LIN {X 0,Y 418.667,Z 234.824,A -85,B 0,C 180,E1 -10080.004,E2 -10080.004} C_VEL
LIN {X 0,Y 418.499,Z 234.849,A -85,B 0,C 180,E1 -10082.892,E2 -10082.892} C_VEL
LIN {X 0,Y 418.499,Z 234.856,A -85,B 0,C 180,E1 -10085.787,E2 -10085.787} C_VEL
LIN {X 0,Y 418.397,Z 234.849,A -85,B 0,C 180,E1 -10088.699,E2 -10088.699} C_VEL
LIN {X 0,Y 418.316,Z 234.859,A -85,B 0,C 180,E1 -10091.635,E2 -10091.635} C_VEL
LIN {X 0,Y 418.306,Z 234.878,A -85,B 0,C 180,E1 -10094.601,E2 -10094.601} C_VEL
LIN {X 0,Y 418.29,Z 234.876,A -85,B 0,C 180,E1 -10097.607,E2 -10097.607} C_VEL
LIN {X 0,Y 418.255,Z 234.87,A -85,B 0,C 180,E1 -10100.666,E2 -10100.666} C_VEL
LIN {X 0,Y 418.28,Z 234.875,A -85,B 0,C 180,E1 -10103.785,E2 -10103.785} C_VEL
LIN {X 0,Y 418.317,Z 234.875,A -85,B 0,C 180,E1 -10107.073,E2 -10107.073} C_VEL
LIN {X 0,Y 418.251,Z 234.871,A -85,B 0,C 180,E1 -10110.275,E2 -10110.275} C_VEL
LIN {X 0,Y 418.24,Z 234.886,A -85,B 0,C 180,E1 -10113.681,E2 -10113.681} C_VEL
LIN {X 0,Y 418.246,Z 234.881,A -85,B 0,C 180,E1 -10117.227,E2 -10117.227} C_VEL
LIN {X 0,Y 418.237,Z 234.887,A -85,B 0,C 180,E1 -10119.687,E2 -10119.687} C_VEL
LIN {X 0,Y 418.232,Z 234.879,A -85,B 0,C 180,E1 -10122.322,E2 -10122.322} C_VEL
LIN {X 0,Y 418.245,Z 234.862,A -85,B 0,C 180,E1 -10125.111,E2 -10125.111} C_VEL
LIN {X 0,Y 418.243,Z 234.883,A -85,B 0,C 180,E1 -10127.768,E2 -10127.768} C_VEL
LIN {X 0,Y 418.247,Z 234.881,A -85,B 0,C 180,E1 -10131.558,E2 -10131.558} C_VEL
LIN {X 0,Y 418.269,Z 234.881,A -85,B 0,C 180,E1 -10135.16,E2 -10135.16} C_VEL
LIN {X 0,Y 418.255,Z 234.885,A -85,B 0,C 180,E1 -10137.473,E2 -10137.473} C_VEL
LIN {X 0,Y 418.279,Z 234.882,A -85,B 0,C 180,E1 -10140.897,E2 -10140.897} C_VEL
LIN {X 0,Y 418.338,Z 234.979,A -85,B 0,C 180,E1 -10143.833,E2 -10143.833} C_VEL
LIN {X 0,Y 419.166,Z 239.348,A -85,B 0,C 180,E1 -10144.881,E2 -10144.881} C_VEL
LIN {X 0,Y 420.709,Z 247.766,A -85,B 0,C 180,E1 -10146.753,E2 -10146.753} C_VEL
LIN {X 0,Y 420.134,Z 259.403,A -85,B 0,C 180,E1 -10149.178,E2 -10149.178} C_VEL
LIN {X 0,Y 419.569,Z 269.337,A -85,B 0,C 180,E1 -10151.189,E2 -10151.189} C_VEL
LIN {X 0,Y 420.301,Z 274.486,A -85,B 0,C 180,E1 -10151.353,E2 -10151.353} C_VEL
LIN {X 0,Y 423.345,Z 294.383,A -85,B 0,C 180,E1 -10151.82,E2 -10151.82} C_VEL
LIN {X 0,Y 422.372,Z 377.264,A -85,B 0,C 180,E1 -10153.258,E2 -10153.258} C_VEL
LIN {X 0,Y 421.886,Z 390.497,A -85,B 0,C 180,E1 -10153.674,E2 -10153.674} C_VEL
LIN {X 0,Y 421.378,Z 403.241,A -85,B 0,C 180,E1 -10154.275,E2 -10154.275} C_VEL
LIN {X 0,Y 420.699,Z 414.545,A -85,B 0,C 180,E1 -10154.993,E2 -10154.993} C_VEL
LIN {X 0,Y 419.998,Z 426.666,A -85,B 0,C 180,E1 -10155.999,E2 -10155.999} C_VEL
LIN {X 0,Y 419.321,Z 437.803,A -85,B 0,C 180,E1 -10157.169,E2 -10157.169} C_VEL
LIN {X 0,Y 418.652,Z 447.013,A -85,B 0,C 180,E1 -10158.379,E2 -10158.379} C_VEL
LIN {X 0,Y 418.063,Z 455.979,A -85,B 0,C 180,E1 -10159.834,E2 -10159.834} C_VEL
LIN {X 0,Y 417.61,Z 463.179,A -85,B 0,C 180,E1 -10161.289,E2 -10161.289} C_VEL
LIN {X 0,Y 417.295,Z 468.908,A -85,B 0,C 180,E1 -10162.744,E2 -10162.744} C_VEL
LIN {X 0,Y 417.132,Z 473.414,A -85,B 0,C 180,E1 -10164.198,E2 -10164.198} C_VEL
LIN {X 0,Y 417.119,Z 475.788,A -85,B 0,C 180,E1 -10165.168,E2 -10165.168} C_VEL
LIN {X 0,Y 417.003,Z 477.727,A -85,B 0,C 180,E1 -10166.135,E2 -10166.135} C_VEL
LIN {X 0,Y 416.988,Z 479.244,A -85,B 0,C 180,E1 -10167.102,E2 -10167.102} C_VEL
LIN {X 0,Y 417.034,Z 480.308,A -85,B 0,C 180,E1 -10168.069,E2 -10168.069} C_VEL
LIN {X 0,Y 416.987,Z 481.258,A -85,B 0,C 180,E1 -10170,E2 -10170} C_VEL
LIN {X 0,Y 416.997,Z 481.151,A -85,B 0,C 180,E1 -10170.966,E2 -10170.966} C_VEL
LIN {X 0,Y 417.035,Z 480.612,A -85,B 0,C 180,E1 -10171.932,E2 -10171.932} C_VEL
LIN {X 0,Y 417.005,Z 478.355,A -85,B 0,C 180,E1 -10173.866,E2 -10173.866} C_VEL
LIN {X 0,Y 417.164,Z 475.557,A -85,B 0,C 180,E1 -10175.317,E2 -10175.317} C_VEL
LIN {X 0,Y 417.253,Z 471.743,A -85,B 0,C 180,E1 -10176.771,E2 -10176.771} C_VEL
LIN {X 0,Y 417.556,Z 466.815,A -85,B 0,C 180,E1 -10178.226,E2 -10178.226} C_VEL
LIN {X 0,Y 418.02,Z 460.625,A -85,B 0,C 180,E1 -10179.679,E2 -10179.679} C_VEL
LIN {X 0,Y 418.572,Z 452.92,A -85,B 0,C 180,E1 -10181.133,E2 -10181.133} C_VEL
LIN {X 0,Y 419.415,Z 443.274,A -85,B 0,C 180,E1 -10182.582,E2 -10182.582} C_VEL
LIN {X 0,Y 420.131,Z 434.12,A -85,B 0,C 180,E1 -10183.7,E2 -10183.7} C_VEL
LIN {X 0,Y 420.84,Z 423.528,A -85,B 0,C 180,E1 -10184.755,E2 -10184.755} C_VEL
LIN {X 0,Y 421.759,Z 411.13,A -85,B 0,C 180,E1 -10185.711,E2 -10185.711} C_VEL
LIN {X 0,Y 422.466,Z 398.984,A -85,B 0,C 180,E1 -10186.428,E2 -10186.428} C_VEL
LIN {X 0,Y 423.138,Z 386.274,A -85,B 0,C 180,E1 -10186.96,E2 -10186.96} C_VEL
LIN {X 0,Y 423.537,Z 372.944,A -85,B 0,C 180,E1 -10187.317,E2 -10187.317} C_VEL
LIN {X 0,Y 424.436,Z 292.84,A -85,B 0,C 180,E1 -10188.717,E2 -10188.717} C_VEL
LIN {X 0,Y 420.28,Z 270.162,A -85,B 0,C 180,E1 -10189.361,E2 -10189.361} C_VEL
LIN {X 0,Y 420.136,Z 269.165,A -85,B 0,C 180,E1 -10189.42,E2 -10189.42} C_VEL
LIN {X 0,Y 421.124,Z 253.902,A -85,B 0,C 180,E1 -10192.572,E2 -10192.572} C_VEL
LIN {X 0,Y 421.179,Z 249.106,A -85,B 0,C 180,E1 -10193.608,E2 -10193.608} C_VEL
LIN {X 0,Y 418.823,Z 237.22,A -85,B 0,C 180,E1 -10196.403,E2 -10196.403} C_VEL
LIN {X 0,Y 418.321,Z 234.928,A -85,B 0,C 180,E1 -10197.026,E2 -10197.026} C_VEL
LIN {X 0,Y 418.257,Z 234.884,A -85,B 0,C 180,E1 -10200.271,E2 -10200.271} C_VEL
LIN {X 0,Y 418.261,Z 234.882,A -85,B 0,C 180,E1 -10203.676,E2 -10203.676} C_VEL
LIN {X 0,Y 418.25,Z 234.885,A -85,B 0,C 180,E1 -10207.223,E2 -10207.223} C_VEL
LIN {X 0,Y 418.222,Z 234.888,A -85,B 0,C 180,E1 -10210.866,E2 -10210.866} C_VEL
LIN {X 0,Y 418.219,Z 234.883,A -85,B 0,C 180,E1 -10213.727,E2 -10213.727} C_VEL
LIN {X 0,Y 418.219,Z 234.881,A -85,B 0,C 180,E1 -10216.447,E2 -10216.447} C_VEL
LIN {X 0,Y 418.229,Z 234.887,A -85,B 0,C 180,E1 -10219.129,E2 -10219.129} C_VEL
LIN {X 0,Y 418.233,Z 234.884,A -85,B 0,C 180,E1 -10222.166,E2 -10222.166} C_VEL
LIN {X 0,Y 418.264,Z 234.882,A -85,B 0,C 180,E1 -10225.42,E2 -10225.42} C_VEL
LIN {X 0,Y 418.221,Z 234.885,A -85,B 0,C 180,E1 -10228.601,E2 -10228.601} C_VEL
LIN {X 0,Y 418.272,Z 234.883,A -85,B 0,C 180,E1 -10230.895,E2 -10230.895} C_VEL
LIN {X 0,Y 418.228,Z 234.885,A -85,B 0,C 180,E1 -10234.09,E2 -10234.09} C_VEL
LIN {X 0,Y 418.237,Z 234.889,A -85,B 0,C 180,E1 -10237.26,E2 -10237.26} C_VEL
LIN {X 0,Y 418.292,Z 234.872,A -85,B 0,C 180,E1 -10240.361,E2 -10240.361} C_VEL
LIN {X 0,Y 418.324,Z 234.875,A -85,B 0,C 180,E1 -10243.401,E2 -10243.401} C_VEL
LIN {X 0,Y 418.353,Z 234.871,A -85,B 0,C 180,E1 -10246.996,E2 -10246.996} C_VEL
LIN {X 0,Y 418.341,Z 234.871,A -85,B 0,C 180,E1 -10250.325,E2 -10250.325} C_VEL
LIN {X 0,Y 418.47,Z 234.854,A -85,B 0,C 180,E1 -10253.245,E2 -10253.245} C_VEL
LIN {X 0,Y 418.329,Z 234.871,A -85,B 0,C 180,E1 -10255.177,E2 -10255.177} C_VEL
LIN {X 0,Y 418.54,Z 234.845,A -85,B 0,C 180,E1 -10258.071,E2 -10258.071} C_VEL
LIN {X 0,Y 418.667,Z 234.833,A -85,B 0,C 180,E1 -10259.996,E2 -10259.996} C_VEL
LIN {X 0,Y 418.491,Z 234.846,A -85,B 0,C 180,E1 -10262.883,E2 -10262.883} C_VEL
LIN {X 0,Y 418.455,Z 234.853,A -85,B 0,C 180,E1 -10266.511,E2 -10266.511} C_VEL
LIN {X 0,Y 418.334,Z 234.873,A -85,B 0,C 180,E1 -10269.667,E2 -10269.667} C_VEL
LIN {X 0,Y 418.339,Z 234.874,A -85,B 0,C 180,E1 -10272.996,E2 -10272.996} C_VEL
LIN {X 0,Y 418.302,Z 234.883,A -85,B 0,C 180,E1 -10276.73,E2 -10276.73} C_VEL
LIN {X 0,Y 418.259,Z 234.881,A -85,B 0,C 180,E1 -10279.785,E2 -10279.785} C_VEL
LIN {X 0,Y 418.224,Z 234.888,A -85,B 0,C 180,E1 -10282.731,E2 -10282.731} C_VEL
LIN {X 0,Y 418.254,Z 234.87,A -85,B 0,C 180,E1 -10285.899,E2 -10285.899} C_VEL
LIN {X 0,Y 418.246,Z 234.887,A -85,B 0,C 180,E1 -10289.157,E2 -10289.157} C_VEL
LIN {X 0,Y 418.235,Z 234.887,A -85,B 0,C 180,E1 -10292.839,E2 -10292.839} C_VEL
LIN {X 0,Y 418.224,Z 234.887,A -85,B 0,C 180,E1 -10296.234,E2 -10296.234} C_VEL
LIN {X 0,Y 418.24,Z 234.889,A -85,B 0,C 180,E1 -10299.675,E2 -10299.675} C_VEL
LIN {X 0,Y 418.256,Z 234.885,A -85,B 0,C 180,E1 -10302.325,E2 -10302.325} C_VEL
LIN {X 0,Y 418.243,Z 234.885,A -85,B 0,C 180,E1 -10305.11,E2 -10305.11} C_VEL
LIN {X 0,Y 418.27,Z 235,A -85,B 0,C 180,E1 -10307.246,E2 -10307.246} C_VEL
LIN {X 0,Y 420.332,Z 244.772,A -85,B 0,C 180,E1 -10309.65,E2 -10309.65} C_VEL
LIN {X 0,Y 420.779,Z 248.927,A -85,B 0,C 180,E1 -10310.603,E2 -10310.603} C_VEL
LIN {X 0,Y 420.313,Z 258.414,A -85,B 0,C 180,E1 -10312.616,E2 -10312.616} C_VEL
LIN {X 0,Y 420.972,Z 261.749,A -85,B 0,C 180,E1 -10312.767,E2 -10312.767} C_VEL
LIN {X 0,Y 424.636,Z 280.212,A -85,B 0,C 180,E1 -10313.303,E2 -10313.303} C_VEL
LIN {X 0,Y 423.482,Z 366.216,A -85,B 0,C 180,E1 -10314.817,E2 -10314.817} C_VEL
LIN {X 0,Y 423.035,Z 379.546,A -85,B 0,C 180,E1 -10315.247,E2 -10315.247} C_VEL
LIN {X 0,Y 422.421,Z 392.479,A -85,B 0,C 180,E1 -10315.867,E2 -10315.867} C_VEL
LIN {X 0,Y 421.668,Z 404.168,A -85,B 0,C 180,E1 -10316.632,E2 -10316.632} C_VEL
LIN {X 0,Y 420.961,Z 415.232,A -85,B 0,C 180,E1 -10317.566,E2 -10317.566} C_VEL
LIN {X 0,Y 420.165,Z 425.427,A -85,B 0,C 180,E1 -10318.634,E2 -10318.634} C_VEL
LIN {X 0,Y 419.394,Z 434.614,A -85,B 0,C 180,E1 -10319.819,E2 -10319.819} C_VEL
LIN {X 0,Y 418.71,Z 442.951,A -85,B 0,C 180,E1 -10321.147,E2 -10321.147} C_VEL
LIN {X 0,Y 418.037,Z 450.97,A -85,B 0,C 180,E1 -10322.734,E2 -10322.734} C_VEL
LIN {X 0,Y 417.66,Z 456.306,A -85,B 0,C 180,E1 -10324.055,E2 -10324.055} C_VEL
LIN {X 0,Y 417.323,Z 461.763,A -85,B 0,C 180,E1 -10325.773,E2 -10325.773} C_VEL
LIN {X 0,Y 417.131,Z 465.133,A -85,B 0,C 180,E1 -10327.2,E2 -10327.2} C_VEL
LIN {X 0,Y 417.012,Z 466.956,A -85,B 0,C 180,E1 -10328.237,E2 -10328.237} C_VEL
LIN {X 0,Y 416.918,Z 468.317,A -85,B 0,C 180,E1 -10329.268,E2 -10329.268} C_VEL
LIN {X 0,Y 416.896,Z 469.449,A -85,B 0,C 180,E1 -10330.721,E2 -10330.721} C_VEL
LIN {X 0,Y 416.836,Z 469.663,A -85,B 0,C 180,E1 -10332.333,E2 -10332.333} C_VEL
LIN {X 0,Y 416.888,Z 468.808,A -85,B 0,C 180,E1 -10333.904,E2 -10333.904} C_VEL
LIN {X 0,Y 416.945,Z 467.072,A -85,B 0,C 180,E1 -10335.354,E2 -10335.354} C_VEL
LIN {X 0,Y 417.113,Z 464.287,A -85,B 0,C 180,E1 -10336.852,E2 -10336.852} C_VEL
LIN {X 0,Y 417.3,Z 460.446,A -85,B 0,C 180,E1 -10338.34,E2 -10338.34} C_VEL
LIN {X 0,Y 417.51,Z 455.46,A -85,B 0,C 180,E1 -10339.819,E2 -10339.819} C_VEL
LIN {X 0,Y 417.941,Z 449.163,A -85,B 0,C 180,E1 -10341.295,E2 -10341.295} C_VEL
LIN {X 0,Y 418.086,Z 446.792,A -85,B 0,C 180,E1 -10341.771,E2 -10341.771} C_VEL
LIN {X 0,Y 417.631,Z 443.355,A -85,B 0,C 180,E1 -10342.428,E2 -10342.428} C_VEL
LIN {X 0,Y 415.128,Z 437.444,A -85,B 0,C 180,E1 -10343.472,E2 -10343.472} C_VEL
LIN {X 0,Y 412.715,Z 430.992,A -85,B 0,C 180,E1 -10344.46,E2 -10344.46} C_VEL
LIN {X 0,Y 412.398,Z 426.689,A -85,B 0,C 180,E1 -10345.022,E2 -10345.022} C_VEL
LIN {X 0,Y 413.087,Z 416.842,A -85,B 0,C 180,E1 -10346.098,E2 -10346.098} C_VEL
LIN {X 0,Y 413.824,Z 405.576,A -85,B 0,C 180,E1 -10347.079,E2 -10347.079} C_VEL
LIN {X 0,Y 414.478,Z 394.904,A -85,B 0,C 180,E1 -10347.813,E2 -10347.813} C_VEL
LIN {X 0,Y 414.954,Z 382.663,A -85,B 0,C 180,E1 -10348.46,E2 -10348.46} C_VEL
LIN {X 0,Y 415.414,Z 369.846,A -85,B 0,C 180,E1 -10348.924,E2 -10348.924} C_VEL
LIN {X 0,Y 415.704,Z 352.192,A -85,B 0,C 180,E1 -10349.288,E2 -10349.288} C_VEL
LIN {X 0,Y 416.536,Z 280.322,A -85,B 0,C 180,E1 -10350.528,E2 -10350.528} C_VEL
LIN {X 0,Y 412.932,Z 260.32,A -85,B 0,C 180,E1 -10351.036,E2 -10351.036} C_VEL
LIN {X 0,Y 412.743,Z 258.407,A -85,B 0,C 180,E1 -10351.158,E2 -10351.158} C_VEL
LIN {X 0,Y 413.343,Z 247.17,A -85,B 0,C 180,E1 -10353.655,E2 -10353.655} C_VEL
LIN {X 0,Y 411.469,Z 235.92,A -85,B 0,C 180,E1 -10356.374,E2 -10356.374} C_VEL
LIN {X 0,Y 411.319,Z 235.75,A -85,B 0,C 180,E1 -10359.838,E2 -10359.838} C_VEL
LIN {X 0,Y 411.333,Z 235.747,A -85,B 0,C 180,E1 -10363.151,E2 -10363.151} C_VEL
LIN {X 0,Y 411.254,Z 235.757,A -85,B 0,C 180,E1 -10366.888,E2 -10366.888} C_VEL
LIN {X 0,Y 411.212,Z 235.748,A -85,B 0,C 180,E1 -10369.987,E2 -10369.987} C_VEL
LIN {X 0,Y 411.201,Z 235.764,A -85,B 0,C 180,E1 -10373.147,E2 -10373.147} C_VEL
LIN {X 0,Y 411.195,Z 235.742,A -85,B 0,C 180,E1 -10376.383,E2 -10376.383} C_VEL
LIN {X 0,Y 411.208,Z 235.761,A -85,B 0,C 180,E1 -10379.712,E2 -10379.712} C_VEL
LIN {X 0,Y 411.214,Z 235.765,A -85,B 0,C 180,E1 -10383.155,E2 -10383.155} C_VEL
LIN {X 0,Y 411.198,Z 235.757,A -85,B 0,C 180,E1 -10386.741,E2 -10386.741} C_VEL
LIN {X 0,Y 411.2,Z 235.763,A -85,B 0,C 180,E1 -10389.736,E2 -10389.736} C_VEL
LIN {X 0,Y 411.196,Z 235.749,A -85,B 0,C 180,E1 -10393.13,E2 -10393.13} C_VEL
LIN {X 0,Y 411.215,Z 235.763,A -85,B 0,C 180,E1 -10395.874,E2 -10395.874} C_VEL
LIN {X 0,Y 411.183,Z 235.759,A -85,B 0,C 180,E1 -10399.504,E2 -10399.504} C_VEL
LIN {X 0,Y 411.177,Z 235.75,A -85,B 0,C 180,E1 -10402.032,E2 -10402.032} C_VEL
LIN {X 0,Y 411.18,Z 235.762,A -85,B 0,C 180,E1 -10405.671,E2 -10405.671} C_VEL
LIN {X 0,Y 411.177,Z 235.757,A -85,B 0,C 180,E1 -10409.158,E2 -10409.158} C_VEL
LIN {X 0,Y 411.238,Z 235.738,A -85,B 0,C 180,E1 -10412.527,E2 -10412.527} C_VEL
LIN {X 0,Y 411.209,Z 235.754,A -85,B 0,C 180,E1 -10415.79,E2 -10415.79} C_VEL
LIN {X 0,Y 411.216,Z 235.763,A -85,B 0,C 180,E1 -10418.973,E2 -10418.973} C_VEL
LIN {X 0,Y 411.238,Z 235.746,A -85,B 0,C 180,E1 -10422.09,E2 -10422.09} C_VEL
LIN {X 0,Y 411.25,Z 235.733,A -85,B 0,C 180,E1 -10425.152,E2 -10425.152} C_VEL
LIN {X 0,Y 411.29,Z 235.742,A -85,B 0,C 180,E1 -10428.172,E2 -10428.172} C_VEL
LIN {X 0,Y 411.474,Z 235.725,A -85,B 0,C 180,E1 -10432.151,E2 -10432.151} C_VEL
LIN {X 0,Y 411.47,Z 235.72,A -85,B 0,C 180,E1 -10434.123,E2 -10434.123} C_VEL
LIN {X 0,Y 411.507,Z 235.701,A -85,B 0,C 180,E1 -10438.047,E2 -10438.047} C_VEL
LIN {X 0,Y 411.637,Z 235.699,A -85,B 0,C 180,E1 -10440.004,E2 -10440.004} C_VEL
LIN {X 0,Y 411.456,Z 235.727,A -85,B 0,C 180,E1 -10442.942,E2 -10442.942} C_VEL
LIN {X 0,Y 411.424,Z 235.727,A -85,B 0,C 180,E1 -10446.872,E2 -10446.872} C_VEL
LIN {X 0,Y 411.293,Z 235.732,A -85,B 0,C 180,E1 -10449.843,E2 -10449.843} C_VEL
LIN {X 0,Y 411.308,Z 235.741,A -85,B 0,C 180,E1 -10453.108,E2 -10453.108} C_VEL
LIN {X 0,Y 411.261,Z 235.752,A -85,B 0,C 180,E1 -10456.892,E2 -10456.892} C_VEL
LIN {X 0,Y 411.236,Z 235.748,A -85,B 0,C 180,E1 -10459.99,E2 -10459.99} C_VEL
LIN {X 0,Y 411.201,Z 235.759,A -85,B 0,C 180,E1 -10463.151,E2 -10463.151} C_VEL
LIN {X 0,Y 411.24,Z 235.76,A -85,B 0,C 180,E1 -10466.384,E2 -10466.384} C_VEL
LIN {X 0,Y 411.208,Z 235.747,A -85,B 0,C 180,E1 -10469.716,E2 -10469.716} C_VEL
LIN {X 0,Y 411.212,Z 235.766,A -85,B 0,C 180,E1 -10473.159,E2 -10473.159} C_VEL
LIN {X 0,Y 411.2,Z 235.758,A -85,B 0,C 180,E1 -10476.555,E2 -10476.555} C_VEL
LIN {X 0,Y 411.204,Z 235.762,A -85,B 0,C 180,E1 -10479.727,E2 -10479.727} C_VEL
LIN {X 0,Y 411.179,Z 235.756,A -85,B 0,C 180,E1 -10483.136,E2 -10483.136} C_VEL
LIN {X 0,Y 411.177,Z 235.746,A -85,B 0,C 180,E1 -10485.883,E2 -10485.883} C_VEL
LIN {X 0,Y 411.167,Z 235.764,A -85,B 0,C 180,E1 -10488.775,E2 -10488.775} C_VEL
LIN {X 0,Y 411.195,Z 235.758,A -85,B 0,C 180,E1 -10492.027,E2 -10492.027} C_VEL
LIN {X 0,Y 411.215,Z 235.76,A -85,B 0,C 180,E1 -10495.668,E2 -10495.668} C_VEL
LIN {X 0,Y 411.2,Z 235.762,A -85,B 0,C 180,E1 -10499.154,E2 -10499.154} C_VEL
LIN {X 0,Y 411.267,Z 235.756,A -85,B 0,C 180,E1 -10502.703,E2 -10502.703} C_VEL
LIN {X 0,Y 411.318,Z 235.847,A -85,B 0,C 180,E1 -10503.625,E2 -10503.625} C_VEL
LIN {X 0,Y 412.71,Z 243.082,A -85,B 0,C 180,E1 -10505.342,E2 -10505.342} C_VEL
LIN {X 0,Y 413.741,Z 249.129,A -85,B 0,C 180,E1 -10506.704,E2 -10506.704} C_VEL
LIN {X 0,Y 413.068,Z 261.662,A -85,B 0,C 180,E1 -10509.36,E2 -10509.36} C_VEL
LIN {X 0,Y 412.604,Z 269.388,A -85,B 0,C 180,E1 -10510.924,E2 -10510.924} C_VEL
LIN {X 0,Y 414.024,Z 278.797,A -85,B 0,C 180,E1 -10511.185,E2 -10511.185} C_VEL
LIN {X 0,Y 416.488,Z 294.407,A -85,B 0,C 180,E1 -10511.558,E2 -10511.558} C_VEL
LIN {X 0,Y 415.539,Z 376.819,A -85,B 0,C 180,E1 -10513.006,E2 -10513.006} C_VEL
LIN {X 0,Y 415.038,Z 390.169,A -85,B 0,C 180,E1 -10513.428,E2 -10513.428} C_VEL
LIN {X 0,Y 414.469,Z 403.532,A -85,B 0,C 180,E1 -10514.069,E2 -10514.069} C_VEL
LIN {X 0,Y 413.719,Z 415.52,A -85,B 0,C 180,E1 -10514.86,E2 -10514.86} C_VEL
LIN {X 0,Y 413.003,Z 427.037,A -85,B 0,C 180,E1 -10515.843,E2 -10515.843} C_VEL
LIN {X 0,Y 412.291,Z 437.367,A -85,B 0,C 180,E1 -10516.947,E2 -10516.947} C_VEL
LIN {X 0,Y 411.668,Z 446.649,A -85,B 0,C 180,E1 -10518.179,E2 -10518.179} C_VEL
LIN {X 0,Y 411.019,Z 455.658,A -85,B 0,C 180,E1 -10519.657,E2 -10519.657} C_VEL
LIN {X 0,Y 410.572,Z 462.905,A -85,B 0,C 180,E1 -10521.138,E2 -10521.138} C_VEL
LIN {X 0,Y 410.216,Z 468.678,A -85,B 0,C 180,E1 -10522.618,E2 -10522.618} C_VEL
LIN {X 0,Y 410.047,Z 473.216,A -85,B 0,C 180,E1 -10524.098,E2 -10524.098} C_VEL
LIN {X 0,Y 410.033,Z 475.604,A -85,B 0,C 180,E1 -10525.084,E2 -10525.084} C_VEL
LIN {X 0,Y 409.924,Z 477.557,A -85,B 0,C 180,E1 -10526.068,E2 -10526.068} C_VEL
LIN {X 0,Y 409.887,Z 479.093,A -85,B 0,C 180,E1 -10527.052,E2 -10527.052} C_VEL
LIN {X 0,Y 409.931,Z 480.177,A -85,B 0,C 180,E1 -10528.035,E2 -10528.035} C_VEL
LIN {X 0,Y 409.923,Z 480.858,A -85,B 0,C 180,E1 -10529.018,E2 -10529.018} C_VEL
LIN {X 0,Y 409.923,Z 481.063,A -85,B 0,C 180,E1 -10530.983,E2 -10530.983} C_VEL
LIN {X 0,Y 409.931,Z 480.545,A -85,B 0,C 180,E1 -10531.965,E2 -10531.965} C_VEL
LIN {X 0,Y 409.926,Z 478.313,A -85,B 0,C 180,E1 -10533.933,E2 -10533.933} C_VEL
LIN {X 0,Y 410.083,Z 475.541,A -85,B 0,C 180,E1 -10535.409,E2 -10535.409} C_VEL
LIN {X 0,Y 410.191,Z 471.754,A -85,B 0,C 180,E1 -10536.889,E2 -10536.889} C_VEL
LIN {X 0,Y 410.529,Z 466.854,A -85,B 0,C 180,E1 -10538.367,E2 -10538.367} C_VEL
LIN {X 0,Y 411.006,Z 460.697,A -85,B 0,C 180,E1 -10539.846,E2 -10539.846} C_VEL
LIN {X 0,Y 411.578,Z 453.046,A -85,B 0,C 180,E1 -10541.325,E2 -10541.325} C_VEL
LIN {X 0,Y 412.482,Z 443.45,A -85,B 0,C 180,E1 -10542.797,E2 -10542.797} C_VEL
LIN {X 0,Y 413.302,Z 433.508,A -85,B 0,C 180,E1 -10544.032,E2 -10544.032} C_VEL
LIN {X 0,Y 414.007,Z 423.885,A -85,B 0,C 180,E1 -10545.004,E2 -10545.004} C_VEL
LIN {X 0,Y 414.861,Z 413.394,A -85,B 0,C 180,E1 -10545.853,E2 -10545.853} C_VEL
LIN {X 0,Y 415.653,Z 400.803,A -85,B 0,C 180,E1 -10546.642,E2 -10546.642} C_VEL
LIN {X 0,Y 416.337,Z 388.247,A -85,B 0,C 180,E1 -10547.214,E2 -10547.214} C_VEL
LIN {X 0,Y 416.827,Z 375.022,A -85,B 0,C 180,E1 -10547.604,E2 -10547.604} C_VEL
LIN {X 0,Y 417.917,Z 294.415,A -85,B 0,C 180,E1 -10549.037,E2 -10549.037} C_VEL
LIN {X 0,Y 413.899,Z 272.234,A -85,B 0,C 180,E1 -10549.675,E2 -10549.675} C_VEL
LIN {X 0,Y 413.259,Z 268.94,A -85,B 0,C 180,E1 -10549.82,E2 -10549.82} C_VEL
LIN {X 0,Y 414.322,Z 254.057,A -85,B 0,C 180,E1 -10552.963,E2 -10552.963} C_VEL
LIN {X 0,Y 414.338,Z 250.928,A -85,B 0,C 180,E1 -10553.655,E2 -10553.655} C_VEL
LIN {X 0,Y 412.129,Z 239.773,A -85,B 0,C 180,E1 -10556.32,E2 -10556.32} C_VEL
LIN {X 0,Y 411.26,Z 235.793,A -85,B 0,C 180,E1 -10557.373,E2 -10557.373} C_VEL
LIN {X 0,Y 411.213,Z 235.764,A -85,B 0,C 180,E1 -10559.712,E2 -10559.712} C_VEL
LIN {X 0,Y 411.22,Z 235.756,A -85,B 0,C 180,E1 -10563.155,E2 -10563.155} C_VEL
LIN {X 0,Y 411.204,Z 235.765,A -85,B 0,C 180,E1 -10566.551,E2 -10566.551} C_VEL
LIN {X 0,Y 411.182,Z 235.761,A -85,B 0,C 180,E1 -10569.719,E2 -10569.719} C_VEL
LIN {X 0,Y 411.182,Z 235.759,A -85,B 0,C 180,E1 -10573.133,E2 -10573.133} C_VEL
LIN {X 0,Y 411.179,Z 235.765,A -85,B 0,C 180,E1 -10575.88,E2 -10575.88} C_VEL
LIN {X 0,Y 411.17,Z 235.764,A -85,B 0,C 180,E1 -10578.771,E2 -10578.771} C_VEL
LIN {X 0,Y 411.198,Z 235.759,A -85,B 0,C 180,E1 -10582.023,E2 -10582.023} C_VEL
LIN {X 0,Y 411.214,Z 235.762,A -85,B 0,C 180,E1 -10585.121,E2 -10585.121} C_VEL
LIN {X 0,Y 411.175,Z 235.76,A -85,B 0,C 180,E1 -10588,E2 -10588} C_VEL
LIN {X 0,Y 411.186,Z 235.76,A -85,B 0,C 180,E1 -10591.404,E2 -10591.404} C_VEL
LIN {X 0,Y 411.198,Z 235.764,A -85,B 0,C 180,E1 -10594.938,E2 -10594.938} C_VEL
LIN {X 0,Y 411.213,Z 235.76,A -85,B 0,C 180,E1 -10597.91,E2 -10597.91} C_VEL
LIN {X 0,Y 411.228,Z 235.755,A -85,B 0,C 180,E1 -10601.048,E2 -10601.048} C_VEL
LIN {X 0,Y 411.261,Z 235.746,A -85,B 0,C 180,E1 -10604.128,E2 -10604.128} C_VEL
LIN {X 0,Y 411.31,Z 235.75,A -85,B 0,C 180,E1 -10607.162,E2 -10607.162} C_VEL
LIN {X 0,Y 411.294,Z 235.751,A -85,B 0,C 180,E1 -10610.157,E2 -10610.157} C_VEL
LIN {X 0,Y 411.436,Z 235.73,A -85,B 0,C 180,E1 -10613.129,E2 -10613.129} C_VEL
LIN {X 0,Y 411.301,Z 235.746,A -85,B 0,C 180,E1 -10615.095,E2 -10615.095} C_VEL
LIN {X 0,Y 411.509,Z 235.721,A -85,B 0,C 180,E1 -10618.038,E2 -10618.038} C_VEL
LIN {X 0,Y 411.636,Z 235.709,A -85,B 0,C 180,E1 -10619.996,E2 -10619.996} C_VEL
LIN {X 0,Y 411.448,Z 235.723,A -85,B 0,C 180,E1 -10622.933,E2 -10622.933} C_VEL
LIN {X 0,Y 411.419,Z 235.73,A -85,B 0,C 180,E1 -10626.508,E2 -10626.508} C_VEL
LIN {X 0,Y 411.286,Z 235.752,A -85,B 0,C 180,E1 -10629.834,E2 -10629.834} C_VEL
LIN {X 0,Y 411.298,Z 235.75,A -85,B 0,C 180,E1 -10633.099,E2 -10633.099} C_VEL
LIN {X 0,Y 411.253,Z 235.759,A -85,B 0,C 180,E1 -10636.864,E2 -10636.864} C_VEL
LIN {X 0,Y 411.219,Z 235.759,A -85,B 0,C 180,E1 -10639.982,E2 -10639.982} C_VEL
LIN {X 0,Y 411.189,Z 235.767,A -85,B 0,C 180,E1 -10643.142,E2 -10643.142} C_VEL
LIN {X 0,Y 411.221,Z 235.746,A -85,B 0,C 180,E1 -10646.376,E2 -10646.376} C_VEL
LIN {X 0,Y 411.181,Z 235.761,A -85,B 0,C 180,E1 -10649.708,E2 -10649.708} C_VEL
LIN {X 0,Y 411.184,Z 235.769,A -85,B 0,C 180,E1 -10653.151,E2 -10653.151} C_VEL
LIN {X 0,Y 411.171,Z 235.766,A -85,B 0,C 180,E1 -10656.548,E2 -10656.548} C_VEL
LIN {X 0,Y 411.202,Z 235.765,A -85,B 0,C 180,E1 -10659.726,E2 -10659.726} C_VEL
LIN {X 0,Y 411.201,Z 235.762,A -85,B 0,C 180,E1 -10663.121,E2 -10663.121} C_VEL
LIN {X 0,Y 411.21,Z 235.763,A -85,B 0,C 180,E1 -10666.703,E2 -10666.703} C_VEL
LIN {X 0,Y 411.28,Z 236.185,A -85,B 0,C 180,E1 -10667.028,E2 -10667.028} C_VEL
LIN {X 0,Y 413.39,Z 246.063,A -85,B 0,C 180,E1 -10669.467,E2 -10669.467} C_VEL
LIN {X 0,Y 413.886,Z 250.239,A -85,B 0,C 180,E1 -10670.448,E2 -10670.448} C_VEL
LIN {X 0,Y 413.457,Z 258.683,A -85,B 0,C 180,E1 -10672.252,E2 -10672.252} C_VEL
LIN {X 0,Y 417.045,Z 275.416,A -85,B 0,C 180,E1 -10672.803,E2 -10672.803} C_VEL
LIN {X 0,Y 418.024,Z 281.178,A -85,B 0,C 180,E1 -10672.963,E2 -10672.963} C_VEL
LIN {X 0,Y 416.816,Z 366.904,A -85,B 0,C 180,E1 -10674.503,E2 -10674.503} C_VEL
LIN {X 0,Y 416.331,Z 380.016,A -85,B 0,C 180,E1 -10674.937,E2 -10674.937} C_VEL
LIN {X 0,Y 415.665,Z 393.069,A -85,B 0,C 180,E1 -10675.581,E2 -10675.581} C_VEL
LIN {X 0,Y 414.805,Z 405.729,A -85,B 0,C 180,E1 -10676.443,E2 -10676.443} C_VEL
LIN {X 0,Y 414.077,Z 416.511,A -85,B 0,C 180,E1 -10677.392,E2 -10677.392} C_VEL
LIN {X 0,Y 413.23,Z 426.428,A -85,B 0,C 180,E1 -10678.471,E2 -10678.471} C_VEL
LIN {X 0,Y 412.334,Z 436.314,A -85,B 0,C 180,E1 -10679.814,E2 -10679.814} C_VEL
LIN {X 0,Y 411.616,Z 444.365,A -85,B 0,C 180,E1 -10681.161,E2 -10681.161} C_VEL
LIN {X 0,Y 410.947,Z 452.106,A -85,B 0,C 180,E1 -10682.771,E2 -10682.771} C_VEL
LIN {X 0,Y 410.59,Z 457.277,A -85,B 0,C 180,E1 -10684.12,E2 -10684.12} C_VEL
LIN {X 0,Y 410.267,Z 462.109,A -85,B 0,C 180,E1 -10685.724,E2 -10685.724} C_VEL
LIN {X 0,Y 410.094,Z 464.609,A -85,B 0,C 180,E1 -10686.786,E2 -10686.786} C_VEL
LIN {X 0,Y 409.94,Z 466.619,A -85,B 0,C 180,E1 -10687.841,E2 -10687.841} C_VEL
LIN {X 0,Y 409.842,Z 468.089,A -85,B 0,C 180,E1 -10688.893,E2 -10688.893} C_VEL
LIN {X 0,Y 409.796,Z 469.511,A -85,B 0,C 180,E1 -10690.584,E2 -10690.584} C_VEL
LIN {X 0,Y 409.731,Z 469.809,A -85,B 0,C 180,E1 -10692.016,E2 -10692.016} C_VEL
LIN {X 0,Y 409.791,Z 468.987,A -85,B 0,C 180,E1 -10693.799,E2 -10693.799} C_VEL
LIN {X 0,Y 409.831,Z 467.582,A -85,B 0,C 180,E1 -10695.094,E2 -10695.094} C_VEL
LIN {X 0,Y 409.981,Z 464.985,A -85,B 0,C 180,E1 -10696.619,E2 -10696.619} C_VEL
LIN {X 0,Y 410.196,Z 461.339,A -85,B 0,C 180,E1 -10698.135,E2 -10698.135} C_VEL
LIN {X 0,Y 410.41,Z 456.561,A -85,B 0,C 180,E1 -10699.641,E2 -10699.641} C_VEL
LIN {X 0,Y 410.784,Z 450.502,A -85,B 0,C 180,E1 -10701.142,E2 -10701.142} C_VEL
LIN {X 0,Y 411.295,Z 443.356,A -85,B 0,C 180,E1 -10702.564,E2 -10702.564} C_VEL
LIN {X 0,Y 411.813,Z 435.276,A -85,B 0,C 180,E1 -10703.877,E2 -10703.877} C_VEL
LIN {X 0,Y 412.398,Z 426.689,A -85,B 0,C 180,E1 -10705.022,E2 -10705.022} C_VEL
LIN {X 0,Y 412.104,Z 422.227,A -85,B 0,C 180,E1 -10705.561,E2 -10705.561} C_VEL
LIN {X 0,Y 409.816,Z 414.754,A -85,B 0,C 180,E1 -10706.416,E2 -10706.416} C_VEL
LIN {X 0,Y 407.512,Z 406.843,A -85,B 0,C 180,E1 -10707.19,E2 -10707.19} C_VEL
LIN {X 0,Y 407.184,Z 401.696,A -85,B 0,C 180,E1 -10707.595,E2 -10707.595} C_VEL
LIN {X 0,Y 407.835,Z 389.198,A -85,B 0,C 180,E1 -10708.377,E2 -10708.377} C_VEL
LIN {X 0,Y 408.353,Z 376.617,A -85,B 0,C 180,E1 -10708.949,E2 -10708.949} C_VEL
LIN {X 0,Y 408.703,Z 363.886,A -85,B 0,C 180,E1 -10709.322,E2 -10709.322} C_VEL
LIN {X 0,Y 409.631,Z 280.811,A -85,B 0,C 180,E1 -10710.797,E2 -10710.797} C_VEL
LIN {X 0,Y 405.829,Z 259.102,A -85,B 0,C 180,E1 -10711.377,E2 -10711.377} C_VEL
LIN {X 0,Y 405.856,Z 257.032,A -85,B 0,C 180,E1 -10711.756,E2 -10711.756} C_VEL
LIN {X 0,Y 406.366,Z 248.438,A -85,B 0,C 180,E1 -10713.718,E2 -10713.718} C_VEL
LIN {X 0,Y 404.422,Z 236.719,A -85,B 0,C 180,E1 -10716.611,E2 -10716.611} C_VEL
LIN {X 0,Y 404.272,Z 236.627,A -85,B 0,C 180,E1 -10720.011,E2 -10720.011} C_VEL
LIN {X 0,Y 404.274,Z 236.626,A -85,B 0,C 180,E1 -10723.246,E2 -10723.246} C_VEL
LIN {X 0,Y 404.201,Z 236.631,A -85,B 0,C 180,E1 -10727.192,E2 -10727.192} C_VEL
LIN {X 0,Y 404.165,Z 236.627,A -85,B 0,C 180,E1 -10730.351,E2 -10730.351} C_VEL
LIN {X 0,Y 404.15,Z 236.638,A -85,B 0,C 180,E1 -10733.575,E2 -10733.575} C_VEL
LIN {X 0,Y 404.152,Z 236.616,A -85,B 0,C 180,E1 -10736.88,E2 -10736.88} C_VEL
LIN {X 0,Y 404.157,Z 236.636,A -85,B 0,C 180,E1 -10740.284,E2 -10740.284} C_VEL
LIN {X 0,Y 404.134,Z 236.639,A -85,B 0,C 180,E1 -10743.813,E2 -10743.813} C_VEL
LIN {X 0,Y 404.143,Z 236.637,A -85,B 0,C 180,E1 -10746.887,E2 -10746.887} C_VEL
LIN {X 0,Y 404.161,Z 236.636,A -85,B 0,C 180,E1 -10750.092,E2 -10750.092} C_VEL
LIN {X 0,Y 404.17,Z 236.624,A -85,B 0,C 180,E1 -10753.096,E2 -10753.096} C_VEL
LIN {X 0,Y 404.187,Z 236.64,A -85,B 0,C 180,E1 -10755.94,E2 -10755.94} C_VEL
LIN {X 0,Y 404.134,Z 236.636,A -85,B 0,C 180,E1 -10758.645,E2 -10758.645} C_VEL
LIN {X 0,Y 404.133,Z 236.624,A -85,B 0,C 180,E1 -10761.495,E2 -10761.495} C_VEL
LIN {X 0,Y 404.159,Z 236.637,A -85,B 0,C 180,E1 -10764.989,E2 -10764.989} C_VEL
LIN {X 0,Y 404.126,Z 236.641,A -85,B 0,C 180,E1 -10768.559,E2 -10768.559} C_VEL
LIN {X 0,Y 404.176,Z 236.617,A -85,B 0,C 180,E1 -10772.005,E2 -10772.005} C_VEL
LIN {X 0,Y 404.158,Z 236.633,A -85,B 0,C 180,E1 -10775.339,E2 -10775.339} C_VEL
LIN {X 0,Y 404.172,Z 236.64,A -85,B 0,C 180,E1 -10778.588,E2 -10778.588} C_VEL
LIN {X 0,Y 404.199,Z 236.623,A -85,B 0,C 180,E1 -10781.767,E2 -10781.767} C_VEL
LIN {X 0,Y 404.195,Z 236.61,A -85,B 0,C 180,E1 -10784.887,E2 -10784.887} C_VEL
LIN {X 0,Y 404.26,Z 236.618,A -85,B 0,C 180,E1 -10787.964,E2 -10787.964} C_VEL
LIN {X 0,Y 404.426,Z 236.603,A -85,B 0,C 180,E1 -10792.104,E2 -10792.104} C_VEL
LIN {X 0,Y 404.419,Z 236.599,A -85,B 0,C 180,E1 -10794.02,E2 -10794.02} C_VEL
LIN {X 0,Y 404.476,Z 236.576,A -85,B 0,C 180,E1 -10798.013,E2 -10798.013} C_VEL
LIN {X 0,Y 404.606,Z 236.574,A -85,B 0,C 180,E1 -10800.004,E2 -10800.004} C_VEL
LIN {X 0,Y 404.414,Z 236.604,A -85,B 0,C 180,E1 -10802.993,E2 -10802.993} C_VEL
LIN {X 0,Y 404.369,Z 236.606,A -85,B 0,C 180,E1 -10806.992,E2 -10806.992} C_VEL
LIN {X 0,Y 404.258,Z 236.607,A -85,B 0,C 180,E1 -10810.016,E2 -10810.016} C_VEL
LIN {X 0,Y 404.269,Z 236.618,A -85,B 0,C 180,E1 -10813.215,E2 -10813.215} C_VEL
LIN {X 0,Y 404.22,Z 236.629,A -85,B 0,C 180,E1 -10817.011,E2 -10817.011} C_VEL
LIN {X 0,Y 404.169,Z 236.625,A -85,B 0,C 180,E1 -10820.355,E2 -10820.355} C_VEL
LIN {X 0,Y 404.166,Z 236.633,A -85,B 0,C 180,E1 -10823.578,E2 -10823.578} C_VEL
LIN {X 0,Y 404.188,Z 236.635,A -85,B 0,C 180,E1 -10825.77,E2 -10825.77} C_VEL
LIN {X 0,Y 404.202,Z 236.63,A -85,B 0,C 180,E1 -10828.003,E2 -10828.003} C_VEL
LIN {X 0,Y 404.146,Z 236.639,A -85,B 0,C 180,E1 -10831.561,E2 -10831.561} C_VEL
LIN {X 0,Y 404.182,Z 236.64,A -85,B 0,C 180,E1 -10835.02,E2 -10835.02} C_VEL
LIN {X 0,Y 404.151,Z 236.637,A -85,B 0,C 180,E1 -10838.761,E2 -10838.761} C_VEL
LIN {X 0,Y 404.126,Z 236.641,A -85,B 0,C 180,E1 -10841.601,E2 -10841.601} C_VEL
LIN {X 0,Y 404.154,Z 236.617,A -85,B 0,C 180,E1 -10844.524,E2 -10844.524} C_VEL
LIN {X 0,Y 404.142,Z 236.631,A -85,B 0,C 180,E1 -10847.297,E2 -10847.297} C_VEL
LIN {X 0,Y 404.143,Z 236.642,A -85,B 0,C 180,E1 -10849.953,E2 -10849.953} C_VEL
LIN {X 0,Y 404.144,Z 236.638,A -85,B 0,C 180,E1 -10853.128,E2 -10853.128} C_VEL
LIN {X 0,Y 404.155,Z 236.639,A -85,B 0,C 180,E1 -10856.189,E2 -10856.189} C_VEL
LIN {X 0,Y 404.156,Z 236.644,A -85,B 0,C 180,E1 -10859.716,E2 -10859.716} C_VEL
LIN {X 0,Y 404.254,Z 236.716,A -85,B 0,C 180,E1 -10863.406,E2 -10863.406} C_VEL
LIN {X 0,Y 405.901,Z 245.206,A -85,B 0,C 180,E1 -10865.447,E2 -10865.447} C_VEL
LIN {X 0,Y 406.791,Z 251.398,A -85,B 0,C 180,E1 -10866.856,E2 -10866.856} C_VEL
LIN {X 0,Y 405.853,Z 266.039,A -85,B 0,C 180,E1 -10870.001,E2 -10870.001} C_VEL
LIN {X 0,Y 405.659,Z 269.118,A -85,B 0,C 180,E1 -10870.618,E2 -10870.618} C_VEL
LIN {X 0,Y 406.149,Z 272.685,A -85,B 0,C 180,E1 -10870.757,E2 -10870.757} C_VEL
LIN {X 0,Y 409.654,Z 295.322,A -85,B 0,C 180,E1 -10871.309,E2 -10871.309} C_VEL
LIN {X 0,Y 408.648,Z 377.364,A -85,B 0,C 180,E1 -10872.775,E2 -10872.775} C_VEL
LIN {X 0,Y 408.105,Z 391.268,A -85,B 0,C 180,E1 -10873.235,E2 -10873.235} C_VEL
LIN {X 0,Y 407.555,Z 403.748,A -85,B 0,C 180,E1 -10873.856,E2 -10873.856} C_VEL
LIN {X 0,Y 406.8,Z 414.864,A -85,B 0,C 180,E1 -10874.596,E2 -10874.596} C_VEL
LIN {X 0,Y 406.091,Z 426.478,A -85,B 0,C 180,E1 -10875.596,E2 -10875.596} C_VEL
LIN {X 0,Y 405.359,Z 436.917,A -85,B 0,C 180,E1 -10876.72,E2 -10876.72} C_VEL
LIN {X 0,Y 404.677,Z 446.284,A -85,B 0,C 180,E1 -10877.972,E2 -10877.972} C_VEL
LIN {X 0,Y 403.997,Z 455.339,A -85,B 0,C 180,E1 -10879.476,E2 -10879.476} C_VEL
LIN {X 0,Y 403.531,Z 462.627,A -85,B 0,C 180,E1 -10880.982,E2 -10880.982} C_VEL
LIN {X 0,Y 403.164,Z 468.444,A -85,B 0,C 180,E1 -10882.488,E2 -10882.488} C_VEL
LIN {X 0,Y 402.95,Z 473.014,A -85,B 0,C 180,E1 -10883.993,E2 -10883.993} C_VEL
LIN {X 0,Y 402.946,Z 475.42,A -85,B 0,C 180,E1 -10884.997,E2 -10884.997} C_VEL
LIN {X 0,Y 402.846,Z 477.387,A -85,B 0,C 180,E1 -10885.999,E2 -10885.999} C_VEL
LIN {X 0,Y 402.789,Z 478.939,A -85,B 0,C 180,E1 -10887,E2 -10887} C_VEL
LIN {X 0,Y 402.828,Z 480.046,A -85,B 0,C 180,E1 -10888.001,E2 -10888.001} C_VEL
LIN {X 0,Y 402.851,Z 480.741,A -85,B 0,C 180,E1 -10889.001,E2 -10889.001} C_VEL
LIN {X 0,Y 402.851,Z 480.972,A -85,B 0,C 180,E1 -10891,E2 -10891} C_VEL
LIN {X 0,Y 402.827,Z 480.477,A -85,B 0,C 180,E1 -10892,E2 -10892} C_VEL
LIN {X 0,Y 402.85,Z 478.271,A -85,B 0,C 180,E1 -10894.002,E2 -10894.002} C_VEL
LIN {X 0,Y 402.983,Z 475.524,A -85,B 0,C 180,E1 -10895.505,E2 -10895.505} C_VEL
LIN {X 0,Y 403.117,Z 471.767,A -85,B 0,C 180,E1 -10897.01,E2 -10897.01} C_VEL
LIN {X 0,Y 403.491,Z 466.904,A -85,B 0,C 180,E1 -10898.514,E2 -10898.514} C_VEL
LIN {X 0,Y 403.974,Z 460.789,A -85,B 0,C 180,E1 -10900.019,E2 -10900.019} C_VEL
LIN {X 0,Y 404.609,Z 453.201,A -85,B 0,C 180,E1 -10901.523,E2 -10901.523} C_VEL
LIN {X 0,Y 405.564,Z 443.678,A -85,B 0,C 180,E1 -10903.019,E2 -10903.019} C_VEL
LIN {X 0,Y 406.436,Z 433.169,A -85,B 0,C 180,E1 -10904.35,E2 -10904.35} C_VEL
LIN {X 0,Y 407.299,Z 422.911,A -85,B 0,C 180,E1 -10905.385,E2 -10905.385} C_VEL
LIN {X 0,Y 408.171,Z 412.187,A -85,B 0,C 180,E1 -10906.248,E2 -10906.248} C_VEL
LIN {X 0,Y 409.044,Z 399.285,A -85,B 0,C 180,E1 -10907.047,E2 -10907.047} C_VEL
LIN {X 0,Y 409.772,Z 386.907,A -85,B 0,C 180,E1 -10907.595,E2 -10907.595} C_VEL
LIN {X 0,Y 410.19,Z 374.147,A -85,B 0,C 180,E1 -10907.963,E2 -10907.963} C_VEL
LIN {X 0,Y 411.221,Z 294.687,A -85,B 0,C 180,E1 -10909.402,E2 -10909.402} C_VEL
LIN {X 0,Y 407.335,Z 273.354,A -85,B 0,C 180,E1 -10910.034,E2 -10910.034} C_VEL
LIN {X 0,Y 406.441,Z 269.033,A -85,B 0,C 180,E1 -10910.203,E2 -10910.203} C_VEL
LIN {X 0,Y 407.276,Z 257.821,A -85,B 0,C 180,E1 -10912.579,E2 -10912.579} C_VEL
LIN {X 0,Y 407.36,Z 252.021,A -85,B 0,C 180,E1 -10913.877,E2 -10913.877} C_VEL
LIN {X 0,Y 404.951,Z 239.973,A -85,B 0,C 180,E1 -10916.823,E2 -10916.823} C_VEL
LIN {X 0,Y 404.226,Z 236.675,A -85,B 0,C 180,E1 -10917.734,E2 -10917.734} C_VEL
LIN {X 0,Y 404.155,Z 236.64,A -85,B 0,C 180,E1 -10921.445,E2 -10921.445} C_VEL
LIN {X 0,Y 404.158,Z 236.64,A -85,B 0,C 180,E1 -10923.811,E2 -10923.811} C_VEL
LIN {X 0,Y 404.147,Z 236.643,A -85,B 0,C 180,E1 -10926.873,E2 -10926.873} C_VEL
LIN {X 0,Y 404.13,Z 236.643,A -85,B 0,C 180,E1 -10930.073,E2 -10930.073} C_VEL
LIN {X 0,Y 404.161,Z 236.633,A -85,B 0,C 180,E1 -10933.081,E2 -10933.081} C_VEL
LIN {X 0,Y 404.159,Z 236.64,A -85,B 0,C 180,E1 -10935.924,E2 -10935.924} C_VEL
LIN {X 0,Y 404.125,Z 236.638,A -85,B 0,C 180,E1 -10938.632,E2 -10938.632} C_VEL
LIN {X 0,Y 404.156,Z 236.636,A -85,B 0,C 180,E1 -10941.492,E2 -10941.492} C_VEL
LIN {X 0,Y 404.185,Z 236.637,A -85,B 0,C 180,E1 -10944.98,E2 -10944.98} C_VEL
LIN {X 0,Y 404.149,Z 236.637,A -85,B 0,C 180,E1 -10948.44,E2 -10948.44} C_VEL
LIN {X 0,Y 404.162,Z 236.641,A -85,B 0,C 180,E1 -10950.86,E2 -10950.86} C_VEL
LIN {X 0,Y 404.163,Z 236.64,A -85,B 0,C 180,E1 -10954.72,E2 -10954.72} C_VEL
LIN {X 0,Y 404.176,Z 236.64,A -85,B 0,C 180,E1 -10957.505,E2 -10957.505} C_VEL
LIN {X 0,Y 404.171,Z 236.631,A -85,B 0,C 180,E1 -10960.704,E2 -10960.704} C_VEL
LIN {X 0,Y 404.229,Z 236.625,A -85,B 0,C 180,E1 -10963.845,E2 -10963.845} C_VEL
LIN {X 0,Y 404.29,Z 236.623,A -85,B 0,C 180,E1 -10966.935,E2 -10966.935} C_VEL
LIN {X 0,Y 404.26,Z 236.626,A -85,B 0,C 180,E1 -10969.984,E2 -10969.984} C_VEL
LIN {X 0,Y 404.386,Z 236.608,A -85,B 0,C 180,E1 -10973.008,E2 -10973.008} C_VEL
LIN {X 0,Y 404.273,Z 236.621,A -85,B 0,C 180,E1 -10975.009,E2 -10975.009} C_VEL
LIN {X 0,Y 404.477,Z 236.596,A -85,B 0,C 180,E1 -10978.004,E2 -10978.004} C_VEL
LIN {X 0,Y 404.606,Z 236.584,A -85,B 0,C 180,E1 -10979.996,E2 -10979.996} C_VEL
LIN {X 0,Y 404.406,Z 236.6,A -85,B 0,C 180,E1 -10982.984,E2 -10982.984} C_VEL
LIN {X 0,Y 404.368,Z 236.609,A -85,B 0,C 180,E1 -10986.503,E2 -10986.503} C_VEL
LIN {X 0,Y 404.261,Z 236.627,A -85,B 0,C 180,E1 -10988.997,E2 -10988.997} C_VEL
LIN {X 0,Y 404.249,Z 236.623,A -85,B 0,C 180,E1 -10992.037,E2 -10992.037} C_VEL
LIN {X 0,Y 404.198,Z 236.631,A -85,B 0,C 180,E1 -10995.113,E2 -10995.113} C_VEL
LIN {X 0,Y 404.194,Z 236.636,A -85,B 0,C 180,E1 -10998.233,E2 -10998.233} C_VEL
LIN {X 0,Y 404.126,Z 236.64,A -85,B 0,C 180,E1 -11001.414,E2 -11001.414} C_VEL
LIN {X 0,Y 404.162,Z 236.638,A -85,B 0,C 180,E1 -11004.66,E2 -11004.66} C_VEL
LIN {X 0,Y 404.177,Z 236.635,A -85,B 0,C 180,E1 -11007.995,E2 -11007.995} C_VEL
LIN {X 0,Y 404.118,Z 236.639,A -85,B 0,C 180,E1 -11011.553,E2 -11011.553} C_VEL
LIN {X 0,Y 404.162,Z 236.634,A -85,B 0,C 180,E1 -11015.011,E2 -11015.011} C_VEL
LIN {X 0,Y 404.138,Z 236.638,A -85,B 0,C 180,E1 -11018.751,E2 -11018.751} C_VEL
LIN {X 0,Y 404.163,Z 236.64,A -85,B 0,C 180,E1 -11021.606,E2 -11021.606} C_VEL
LIN {X 0,Y 404.17,Z 236.64,A -85,B 0,C 180,E1 -11024.525,E2 -11024.525} C_VEL
LIN {X 0,Y 404.193,Z 236.764,A -85,B 0,C 180,E1 -11026.568,E2 -11026.568} C_VEL
LIN {X 0,Y 406.613,Z 248.274,A -85,B 0,C 180,E1 -11029.499,E2 -11029.499} C_VEL
LIN {X 0,Y 407.005,Z 251.578,A -85,B 0,C 180,E1 -11030.29,E2 -11030.29} C_VEL
LIN {X 0,Y 406.624,Z 258.761,A -85,B 0,C 180,E1 -11031.851,E2 -11031.851} C_VEL
LIN {X 0,Y 410.137,Z 274.956,A -85,B 0,C 180,E1 -11032.401,E2 -11032.401} C_VEL
LIN {X 0,Y 411.453,Z 282.428,A -85,B 0,C 180,E1 -11032.619,E2 -11032.619} C_VEL
LIN {X 0,Y 410.168,Z 366.604,A -85,B 0,C 180,E1 -11034.15,E2 -11034.15} C_VEL
LIN {X 0,Y 409.653,Z 380.064,A -85,B 0,C 180,E1 -11034.6,E2 -11034.6} C_VEL
LIN {X 0,Y 409.016,Z 392.751,A -85,B 0,C 180,E1 -11035.232,E2 -11035.232} C_VEL
LIN {X 0,Y 408.163,Z 404.477,A -85,B 0,C 180,E1 -11036.025,E2 -11036.025} C_VEL
LIN {X 0,Y 407.284,Z 416.399,A -85,B 0,C 180,E1 -11037.074,E2 -11037.074} C_VEL
LIN {X 0,Y 406.361,Z 426.808,A -85,B 0,C 180,E1 -11038.226,E2 -11038.226} C_VEL
LIN {X 0,Y 405.473,Z 436.288,A -85,B 0,C 180,E1 -11039.537,E2 -11039.537} C_VEL
LIN {X 0,Y 404.683,Z 444.352,A -85,B 0,C 180,E1 -11040.904,E2 -11040.904} C_VEL
LIN {X 0,Y 403.981,Z 451.998,A -85,B 0,C 180,E1 -11042.514,E2 -11042.514} C_VEL
LIN {X 0,Y 403.486,Z 458.173,A -85,B 0,C 180,E1 -11044.186,E2 -11044.186} C_VEL
LIN {X 0,Y 403.164,Z 462.812,A -85,B 0,C 180,E1 -11045.817,E2 -11045.817} C_VEL
LIN {X 0,Y 402.873,Z 466.469,A -85,B 0,C 180,E1 -11047.585,E2 -11047.585} C_VEL
LIN {X 0,Y 402.78,Z 467.847,A -85,B 0,C 180,E1 -11048.505,E2 -11048.505} C_VEL
LIN {X 0,Y 402.71,Z 469.572,A -85,B 0,C 180,E1 -11050.437,E2 -11050.437} C_VEL
LIN {X 0,Y 402.65,Z 469.932,A -85,B 0,C 180,E1 -11051.689,E2 -11051.689} C_VEL
LIN {X 0,Y 402.645,Z 469.729,A -85,B 0,C 180,E1 -11052.739,E2 -11052.739} C_VEL
LIN {X 0,Y 402.691,Z 469.09,A -85,B 0,C 180,E1 -11053.785,E2 -11053.785} C_VEL
LIN {X 0,Y 402.732,Z 468.044,A -85,B 0,C 180,E1 -11054.825,E2 -11054.825} C_VEL
LIN {X 0,Y 402.798,Z 466.552,A -85,B 0,C 180,E1 -11055.861,E2 -11055.861} C_VEL
LIN {X 0,Y 403.034,Z 463.165,A -85,B 0,C 180,E1 -11057.525,E2 -11057.525} C_VEL
LIN {X 0,Y 403.217,Z 459.272,A -85,B 0,C 180,E1 -11058.946,E2 -11058.946} C_VEL
LIN {X 0,Y 403.546,Z 452.873,A -85,B 0,C 180,E1 -11060.729,E2 -11060.729} C_VEL
LIN {X 0,Y 404.115,Z 445.243,A -85,B 0,C 180,E1 -11062.379,E2 -11062.379} C_VEL
LIN {X 0,Y 404.684,Z 437.157,A -85,B 0,C 180,E1 -11063.768,E2 -11063.768} C_VEL
LIN {X 0,Y 405.405,Z 427.063,A -85,B 0,C 180,E1 -11065.171,E2 -11065.171} C_VEL
LIN {X 0,Y 406.126,Z 417.137,A -85,B 0,C 180,E1 -11066.279,E2 -11066.279} C_VEL
LIN {X 0,Y 406.891,Z 405.904,A -85,B 0,C 180,E1 -11067.277,E2 -11067.277} C_VEL
LIN {X 0,Y 407.184,Z 401.696,A -85,B 0,C 180,E1 -11067.595,E2 -11067.595} C_VEL
LIN {X 0,Y 406.764,Z 398.19,A -85,B 0,C 180,E1 -11067.861,E2 -11067.861} C_VEL
LIN {X 0,Y 404.235,Z 392.736,A -85,B 0,C 180,E1 -11068.301,E2 -11068.301} C_VEL
LIN {X 0,Y 401.67,Z 387.172,A -85,B 0,C 180,E1 -11068.708,E2 -11068.708} C_VEL
LIN {X 0,Y 401.159,Z 383.495,A -85,B 0,C 180,E1 -11068.91,E2 -11068.91} C_VEL
LIN {X 0,Y 401.665,Z 370.6,A -85,B 0,C 180,E1 -11069.404,E2 -11069.404} C_VEL
LIN {X 0,Y 401.957,Z 355.02,A -85,B 0,C 180,E1 -11069.749,E2 -11069.749} C_VEL
LIN {X 0,Y 402.888,Z 282.031,A -85,B 0,C 180,E1 -11071.056,E2 -11071.056} C_VEL
LIN {X 0,Y 398.884,Z 259.034,A -85,B 0,C 180,E1 -11071.678,E2 -11071.678} C_VEL
LIN {X 0,Y 399.385,Z 249.689,A -85,B 0,C 180,E1 -11073.783,E2 -11073.783} C_VEL
LIN {X 0,Y 397.423,Z 237.809,A -85,B 0,C 180,E1 -11076.728,E2 -11076.728} C_VEL
LIN {X 0,Y 397.338,Z 237.491,A -85,B 0,C 180,E1 -11077.112,E2 -11077.112} C_VEL
LIN {X 0,Y 397.241,Z 237.503,A -85,B 0,C 180,E1 -11080.19,E2 -11080.19} C_VEL
LIN {X 0,Y 397.224,Z 237.504,A -85,B 0,C 180,E1 -11083.35,E2 -11083.35} C_VEL
LIN {X 0,Y 397.18,Z 237.506,A -85,B 0,C 180,E1 -11087.178,E2 -11087.178} C_VEL
LIN {X 0,Y 397.118,Z 237.509,A -85,B 0,C 180,E1 -11090.729,E2 -11090.729} C_VEL
LIN {X 0,Y 397.103,Z 237.514,A -85,B 0,C 180,E1 -11094.02,E2 -11094.02} C_VEL
LIN {X 0,Y 397.153,Z 237.489,A -85,B 0,C 180,E1 -11097.393,E2 -11097.393} C_VEL
LIN {X 0,Y 397.118,Z 237.515,A -85,B 0,C 180,E1 -11100.878,E2 -11100.878} C_VEL
LIN {X 0,Y 397.108,Z 237.511,A -85,B 0,C 180,E1 -11104.494,E2 -11104.494} C_VEL
LIN {X 0,Y 397.114,Z 237.516,A -85,B 0,C 180,E1 -11108.273,E2 -11108.273} C_VEL
LIN {X 0,Y 397.122,Z 237.504,A -85,B 0,C 180,E1 -11111.998,E2 -11111.998} C_VEL
LIN {X 0,Y 397.145,Z 237.509,A -85,B 0,C 180,E1 -11115.06,E2 -11115.06} C_VEL
LIN {X 0,Y 397.126,Z 237.516,A -85,B 0,C 180,E1 -11118.011,E2 -11118.011} C_VEL
LIN {X 0,Y 397.081,Z 237.502,A -85,B 0,C 180,E1 -11121.73,E2 -11121.73} C_VEL
LIN {X 0,Y 397.099,Z 237.516,A -85,B 0,C 180,E1 -11125.512,E2 -11125.512} C_VEL
LIN {X 0,Y 397.063,Z 237.515,A -85,B 0,C 180,E1 -11129.123,E2 -11129.123} C_VEL
LIN {X 0,Y 397.173,Z 237.488,A -85,B 0,C 180,E1 -11132.615,E2 -11132.615} C_VEL
LIN {X 0,Y 397.115,Z 237.51,A -85,B 0,C 180,E1 -11135.987,E2 -11135.987} C_VEL
LIN {X 0,Y 397.151,Z 237.509,A -85,B 0,C 180,E1 -11139.698,E2 -11139.698} C_VEL
LIN {X 0,Y 397.168,Z 237.495,A -85,B 0,C 180,E1 -11142.85,E2 -11142.85} C_VEL
LIN {X 0,Y 397.215,Z 237.485,A -85,B 0,C 180,E1 -11146.684,E2 -11146.684} C_VEL
LIN {X 0,Y 397.22,Z 237.502,A -85,B 0,C 180,E1 -11149.814,E2 -11149.814} C_VEL
LIN {X 0,Y 397.357,Z 237.485,A -85,B 0,C 180,E1 -11152.893,E2 -11152.893} C_VEL
LIN {X 0,Y 397.25,Z 237.492,A -85,B 0,C 180,E1 -11154.93,E2 -11154.93} C_VEL
LIN {X 0,Y 397.445,Z 237.451,A -85,B 0,C 180,E1 -11157.978,E2 -11157.978} C_VEL
LIN {X 0,Y 397.575,Z 237.449,A -85,B 0,C 180,E1 -11160.005,E2 -11160.005} C_VEL
LIN {X 0,Y 397.373,Z 237.481,A -85,B 0,C 180,E1 -11163.046,E2 -11163.046} C_VEL
LIN {X 0,Y 397.345,Z 237.486,A -85,B 0,C 180,E1 -11166.096,E2 -11166.096} C_VEL
LIN {X 0,Y 397.243,Z 237.482,A -85,B 0,C 180,E1 -11169.166,E2 -11169.166} C_VEL
LIN {X 0,Y 397.221,Z 237.493,A -85,B 0,C 180,E1 -11172.262,E2 -11172.262} C_VEL
LIN {X 0,Y 397.182,Z 237.506,A -85,B 0,C 180,E1 -11175.396,E2 -11175.396} C_VEL
LIN {X 0,Y 397.165,Z 237.504,A -85,B 0,C 180,E1 -11178.577,E2 -11178.577} C_VEL
LIN {X 0,Y 397.101,Z 237.502,A -85,B 0,C 180,E1 -11181.822,E2 -11181.822} C_VEL
LIN {X 0,Y 397.157,Z 237.511,A -85,B 0,C 180,E1 -11185.515,E2 -11185.515} C_VEL
LIN {X 0,Y 397.124,Z 237.513,A -85,B 0,C 180,E1 -11188.547,E2 -11188.547} C_VEL
LIN {X 0,Y 397.085,Z 237.518,A -85,B 0,C 180,E1 -11192.075,E2 -11192.075} C_VEL
LIN {X 0,Y 397.107,Z 237.515,A -85,B 0,C 180,E1 -11195.502,E2 -11195.502} C_VEL
LIN {X 0,Y 397.108,Z 237.515,A -85,B 0,C 180,E1 -11198.858,E2 -11198.858} C_VEL
LIN {X 0,Y 397.073,Z 237.515,A -85,B 0,C 180,E1 -11202.27,E2 -11202.27} C_VEL
LIN {X 0,Y 397.096,Z 237.494,A -85,B 0,C 180,E1 -11205.071,E2 -11205.071} C_VEL
LIN {X 0,Y 397.071,Z 237.522,A -85,B 0,C 180,E1 -11208.024,E2 -11208.024} C_VEL
LIN {X 0,Y 397.102,Z 237.513,A -85,B 0,C 180,E1 -11211.726,E2 -11211.726} C_VEL
LIN {X 0,Y 397.135,Z 237.514,A -85,B 0,C 180,E1 -11215.508,E2 -11215.508} C_VEL
LIN {X 0,Y 397.089,Z 237.521,A -85,B 0,C 180,E1 -11219.119,E2 -11219.119} C_VEL
LIN {X 0,Y 397.194,Z 237.51,A -85,B 0,C 180,E1 -11222.895,E2 -11222.895} C_VEL
LIN {X 0,Y 397.25,Z 237.737,A -85,B 0,C 180,E1 -11223.255,E2 -11223.255} C_VEL
LIN {X 0,Y 399.663,Z 250.581,A -85,B 0,C 180,E1 -11226.318,E2 -11226.318} C_VEL
LIN {X 0,Y 399.579,Z 255.939,A -85,B 0,C 180,E1 -11227.509,E2 -11227.509} C_VEL
LIN {X 0,Y 398.742,Z 268.882,A -85,B 0,C 180,E1 -11230.301,E2 -11230.301} C_VEL
LIN {X 0,Y 399.028,Z 271.617,A -85,B 0,C 180,E1 -11230.437,E2 -11230.437} C_VEL
LIN {X 0,Y 402.85,Z 296.626,A -85,B 0,C 180,E1 -11231.059,E2 -11231.059} C_VEL
LIN {X 0,Y 401.808,Z 376.635,A -85,B 0,C 180,E1 -11232.505,E2 -11232.505} C_VEL
LIN {X 0,Y 401.276,Z 389.985,A -85,B 0,C 180,E1 -11232.941,E2 -11232.941} C_VEL
LIN {X 0,Y 400.66,Z 402.788,A -85,B 0,C 180,E1 -11233.57,E2 -11233.57} C_VEL
LIN {X 0,Y 399.95,Z 414.15,A -85,B 0,C 180,E1 -11234.326,E2 -11234.326} C_VEL
LIN {X 0,Y 399.235,Z 425.09,A -85,B 0,C 180,E1 -11235.264,E2 -11235.264} C_VEL
LIN {X 0,Y 398.596,Z 434.636,A -85,B 0,C 180,E1 -11236.277,E2 -11236.277} C_VEL
LIN {X 0,Y 397.846,Z 444.103,A -85,B 0,C 180,E1 -11237.503,E2 -11237.503} C_VEL
LIN {X 0,Y 397.151,Z 452.168,A -85,B 0,C 180,E1 -11238.776,E2 -11238.776} C_VEL
LIN {X 0,Y 396.633,Z 460.07,A -85,B 0,C 180,E1 -11240.31,E2 -11240.31} C_VEL
LIN {X 0,Y 396.219,Z 466.367,A -85,B 0,C 180,E1 -11241.842,E2 -11241.842} C_VEL
LIN {X 0,Y 395.948,Z 471.371,A -85,B 0,C 180,E1 -11243.376,E2 -11243.376} C_VEL
LIN {X 0,Y 395.86,Z 475.229,A -85,B 0,C 180,E1 -11244.908,E2 -11244.908} C_VEL
LIN {X 0,Y 395.771,Z 477.211,A -85,B 0,C 180,E1 -11245.927,E2 -11245.927} C_VEL
LIN {X 0,Y 395.696,Z 478.778,A -85,B 0,C 180,E1 -11246.946,E2 -11246.946} C_VEL
LIN {X 0,Y 395.725,Z 479.913,A -85,B 0,C 180,E1 -11247.965,E2 -11247.965} C_VEL
LIN {X 0,Y 395.762,Z 480.622,A -85,B 0,C 180,E1 -11248.983,E2 -11248.983} C_VEL
LIN {X 0,Y 395.766,Z 480.944,A -85,B 0,C 180,E1 -11250,E2 -11250} C_VEL
LIN {X 0,Y 395.762,Z 480.881,A -85,B 0,C 180,E1 -11251.018,E2 -11251.018} C_VEL
LIN {X 0,Y 395.724,Z 480.413,A -85,B 0,C 180,E1 -11252.036,E2 -11252.036} C_VEL
LIN {X 0,Y 395.777,Z 478.237,A -85,B 0,C 180,E1 -11254.073,E2 -11254.073} C_VEL
LIN {X 0,Y 395.887,Z 475.523,A -85,B 0,C 180,E1 -11255.604,E2 -11255.604} C_VEL
LIN {X 0,Y 396.068,Z 471.801,A -85,B 0,C 180,E1 -11257.135,E2 -11257.135} C_VEL
LIN {X 0,Y 396.464,Z 466.973,A -85,B 0,C 180,E1 -11258.666,E2 -11258.666} C_VEL
LIN {X 0,Y 396.961,Z 460.896,A -85,B 0,C 180,E1 -11260.198,E2 -11260.198} C_VEL
LIN {X 0,Y 397.655,Z 453.355,A -85,B 0,C 180,E1 -11261.727,E2 -11261.727} C_VEL
LIN {X 0,Y 398.501,Z 445.66,A -85,B 0,C 180,E1 -11262.995,E2 -11262.995} C_VEL
LIN {X 0,Y 399.331,Z 436.295,A -85,B 0,C 180,E1 -11264.264,E2 -11264.264} C_VEL
LIN {X 0,Y 400.189,Z 425.922,A -85,B 0,C 180,E1 -11265.404,E2 -11265.404} C_VEL
LIN {X 0,Y 401.271,Z 414.408,A -85,B 0,C 180,E1 -11266.405,E2 -11266.405} C_VEL
LIN {X 0,Y 402.163,Z 402.275,A -85,B 0,C 180,E1 -11267.217,E2 -11267.217} C_VEL
LIN {X 0,Y 402.968,Z 388.815,A -85,B 0,C 180,E1 -11267.869,E2 -11267.869} C_VEL
LIN {X 0,Y 403.516,Z 376.296,A -85,B 0,C 180,E1 -11268.271,E2 -11268.271} C_VEL
LIN {X 0,Y 404.648,Z 295.562,A -85,B 0,C 180,E1 -11269.767,E2 -11269.767} C_VEL
LIN {X 0,Y 400.797,Z 274.667,A -85,B 0,C 180,E1 -11270.402,E2 -11270.402} C_VEL
LIN {X 0,Y 399.615,Z 268.85,A -85,B 0,C 180,E1 -11270.635,E2 -11270.635} C_VEL
LIN {X 0,Y 400.63,Z 255.598,A -85,B 0,C 180,E1 -11273.521,E2 -11273.521} C_VEL
LIN {X 0,Y 399.547,Z 248.536,A -85,B 0,C 180,E1 -11275.235,E2 -11275.235} C_VEL
LIN {X 0,Y 397.231,Z 237.793,A -85,B 0,C 180,E1 -11277.995,E2 -11277.995} C_VEL
LIN {X 0,Y 397.134,Z 237.516,A -85,B 0,C 180,E1 -11278.543,E2 -11278.543} C_VEL
LIN {X 0,Y 397.092,Z 237.522,A -85,B 0,C 180,E1 -11282.071,E2 -11282.071} C_VEL
LIN {X 0,Y 397.132,Z 237.511,A -85,B 0,C 180,E1 -11285.502,E2 -11285.502} C_VEL
LIN {X 0,Y 397.106,Z 237.512,A -85,B 0,C 180,E1 -11288.853,E2 -11288.853} C_VEL
LIN {X 0,Y 397.074,Z 237.515,A -85,B 0,C 180,E1 -11292.267,E2 -11292.267} C_VEL
LIN {X 0,Y 397.098,Z 237.519,A -85,B 0,C 180,E1 -11295.067,E2 -11295.067} C_VEL
LIN {X 0,Y 397.073,Z 237.509,A -85,B 0,C 180,E1 -11298.02,E2 -11298.02} C_VEL
LIN {X 0,Y 397.112,Z 237.515,A -85,B 0,C 180,E1 -11301.142,E2 -11301.142} C_VEL
LIN {X 0,Y 397.111,Z 237.517,A -85,B 0,C 180,E1 -11304.499,E2 -11304.499} C_VEL
LIN {X 0,Y 397.088,Z 237.514,A -85,B 0,C 180,E1 -11307.926,E2 -11307.926} C_VEL
LIN {X 0,Y 397.128,Z 237.515,A -85,B 0,C 180,E1 -11310.292,E2 -11310.292} C_VEL
LIN {X 0,Y 397.086,Z 237.52,A -85,B 0,C 180,E1 -11313.734,E2 -11313.734} C_VEL
LIN {X 0,Y 397.108,Z 237.517,A -85,B 0,C 180,E1 -11317.082,E2 -11317.082} C_VEL
LIN {X 0,Y 397.156,Z 237.504,A -85,B 0,C 180,E1 -11320.349,E2 -11320.349} C_VEL
LIN {X 0,Y 397.174,Z 237.507,A -85,B 0,C 180,E1 -11323.55,E2 -11323.55} C_VEL
LIN {X 0,Y 397.236,Z 237.5,A -85,B 0,C 180,E1 -11326.699,E2 -11326.699} C_VEL
LIN {X 0,Y 397.22,Z 237.501,A -85,B 0,C 180,E1 -11329.805,E2 -11329.805} C_VEL
LIN {X 0,Y 397.334,Z 237.486,A -85,B 0,C 180,E1 -11332.883,E2 -11332.883} C_VEL
LIN {X 0,Y 397.244,Z 237.496,A -85,B 0,C 180,E1 -11334.921,E2 -11334.921} C_VEL
LIN {X 0,Y 397.446,Z 237.472,A -85,B 0,C 180,E1 -11337.969,E2 -11337.969} C_VEL
LIN {X 0,Y 397.575,Z 237.46,A -85,B 0,C 180,E1 -11339.995,E2 -11339.995} C_VEL
LIN {X 0,Y 397.34,Z 237.48,A -85,B 0,C 180,E1 -11343.037,E2 -11343.037} C_VEL
LIN {X 0,Y 397.322,Z 237.488,A -85,B 0,C 180,E1 -11346.496,E2 -11346.496} C_VEL
LIN {X 0,Y 397.231,Z 237.502,A -85,B 0,C 180,E1 -11349.157,E2 -11349.157} C_VEL
LIN {X 0,Y 397.212,Z 237.501,A -85,B 0,C 180,E1 -11352.253,E2 -11352.253} C_VEL
LIN {X 0,Y 397.171,Z 237.505,A -85,B 0,C 180,E1 -11355.387,E2 -11355.387} C_VEL
LIN {X 0,Y 397.147,Z 237.512,A -85,B 0,C 180,E1 -11358.568,E2 -11358.568} C_VEL
LIN {X 0,Y 397.084,Z 237.516,A -85,B 0,C 180,E1 -11361.813,E2 -11361.813} C_VEL
LIN {X 0,Y 397.141,Z 237.505,A -85,B 0,C 180,E1 -11365.126,E2 -11365.126} C_VEL
LIN {X 0,Y 397.144,Z 237.512,A -85,B 0,C 180,E1 -11367.771,E2 -11367.771} C_VEL
LIN {X 0,Y 397.058,Z 237.516,A -85,B 0,C 180,E1 -11370.877,E2 -11370.877} C_VEL
LIN {X 0,Y 397.103,Z 237.515,A -85,B 0,C 180,E1 -11374.488,E2 -11374.488} C_VEL
LIN {X 0,Y 397.085,Z 237.515,A -85,B 0,C 180,E1 -11378.269,E2 -11378.269} C_VEL
LIN {X 0,Y 397.128,Z 237.519,A -85,B 0,C 180,E1 -11381.989,E2 -11381.989} C_VEL
LIN {X 0,Y 397.12,Z 237.516,A -85,B 0,C 180,E1 -11385.055,E2 -11385.055} C_VEL
LIN {X 0,Y 397.151,Z 237.666,A -85,B 0,C 180,E1 -11386.211,E2 -11386.211} C_VEL
LIN {X 0,Y 399.578,Z 248.859,A -85,B 0,C 180,E1 -11389.13,E2 -11389.13} C_VEL
LIN {X 0,Y 400.126,Z 252.854,A -85,B 0,C 180,E1 -11390.111,E2 -11390.111} C_VEL
LIN {X 0,Y 399.849,Z 258.78,A -85,B 0,C 180,E1 -11391.417,E2 -11391.417} C_VEL
LIN {X 0,Y 401.121,Z 264.475,A -85,B 0,C 180,E1 -11391.657,E2 -11391.657} C_VEL
LIN {X 0,Y 404.773,Z 282.481,A -85,B 0,C 180,E1 -11392.227,E2 -11392.227} C_VEL
LIN {X 0,Y 403.905,Z 347.788,A -85,B 0,C 180,E1 -11393.425,E2 -11393.425} C_VEL
LIN {X 0,Y 403.481,Z 368.355,A -85,B 0,C 180,E1 -11393.839,E2 -11393.839} C_VEL
LIN {X 0,Y 402.921,Z 381.865,A -85,B 0,C 180,E1 -11394.321,E2 -11394.321} C_VEL
LIN {X 0,Y 402.233,Z 393.778,A -85,B 0,C 180,E1 -11394.949,E2 -11394.949} C_VEL
LIN {X 0,Y 401.328,Z 405.984,A -85,B 0,C 180,E1 -11395.812,E2 -11395.812} C_VEL
LIN {X 0,Y 400.41,Z 417.696,A -85,B 0,C 180,E1 -11396.886,E2 -11396.886} C_VEL
LIN {X 0,Y 399.359,Z 428.415,A -85,B 0,C 180,E1 -11398.133,E2 -11398.133} C_VEL
LIN {X 0,Y 398.496,Z 437.371,A -85,B 0,C 180,E1 -11399.424,E2 -11399.424} C_VEL
LIN {X 0,Y 397.624,Z 445.805,A -85,B 0,C 180,E1 -11400.918,E2 -11400.918} C_VEL
LIN {X 0,Y 396.891,Z 453.243,A -85,B 0,C 180,E1 -11402.587,E2 -11402.587} C_VEL
LIN {X 0,Y 396.393,Z 459.08,A -85,B 0,C 180,E1 -11404.254,E2 -11404.254} C_VEL
LIN {X 0,Y 396.056,Z 463.529,A -85,B 0,C 180,E1 -11405.912,E2 -11405.912} C_VEL
LIN {X 0,Y 395.829,Z 466.45,A -85,B 0,C 180,E1 -11407.39,E2 -11407.39} C_VEL
LIN {X 0,Y 395.633,Z 468.832,A -85,B 0,C 180,E1 -11409.189,E2 -11409.189} C_VEL
LIN {X 0,Y 395.62,Z 469.637,A -85,B 0,C 180,E1 -11410.287,E2 -11410.287} C_VEL
LIN {X 0,Y 395.561,Z 469.987,A -85,B 0,C 180,E1 -11411.348,E2 -11411.348} C_VEL
LIN {X 0,Y 395.55,Z 469.928,A -85,B 0,C 180,E1 -11412.419,E2 -11412.419} C_VEL
LIN {X 0,Y 395.583,Z 469.335,A -85,B 0,C 180,E1 -11413.587,E2 -11413.587} C_VEL
LIN {X 0,Y 395.671,Z 467.088,A -85,B 0,C 180,E1 -11415.601,E2 -11415.601} C_VEL
LIN {X 0,Y 395.922,Z 463.527,A -85,B 0,C 180,E1 -11417.469,E2 -11417.469} C_VEL
LIN {X 0,Y 396.169,Z 458.603,A -85,B 0,C 180,E1 -11419.265,E2 -11419.265} C_VEL
LIN {X 0,Y 396.498,Z 453.035,A -85,B 0,C 180,E1 -11420.82,E2 -11420.82} C_VEL
LIN {X 0,Y 397.038,Z 446.097,A -85,B 0,C 180,E1 -11422.364,E2 -11422.364} C_VEL
LIN {X 0,Y 397.583,Z 438.953,A -85,B 0,C 180,E1 -11423.657,E2 -11423.657} C_VEL
LIN {X 0,Y 398.154,Z 430.392,A -85,B 0,C 180,E1 -11424.936,E2 -11424.936} C_VEL
LIN {X 0,Y 398.97,Z 419.775,A -85,B 0,C 180,E1 -11426.212,E2 -11426.212} C_VEL
LIN {X 0,Y 399.781,Z 409.226,A -85,B 0,C 180,E1 -11427.229,E2 -11427.229} C_VEL
LIN {X 0,Y 400.535,Z 398.151,A -85,B 0,C 180,E1 -11428.077,E2 -11428.077} C_VEL
LIN {X 0,Y 401.094,Z 386.058,A -85,B 0,C 180,E1 -11428.785,E2 -11428.785} C_VEL
LIN {X 0,Y 401.159,Z 383.495,A -85,B 0,C 180,E1 -11428.91,E2 -11428.91} C_VEL
LIN {X 0,Y 400.811,Z 377.902,A -85,B 0,C 180,E1 -11429.176,E2 -11429.176} C_VEL
LIN {X 0,Y 398.39,Z 368.723,A -85,B 0,C 180,E1 -11429.583,E2 -11429.583} C_VEL
LIN {X 0,Y 395.783,Z 359.408,A -85,B 0,C 180,E1 -11429.908,E2 -11429.908} C_VEL
LIN {X 0,Y 395.151,Z 353.597,A -85,B 0,C 180,E1 -11430.042,E2 -11430.042} C_VEL
LIN {X 0,Y 396.061,Z 282.654,A -85,B 0,C 180,E1 -11431.337,E2 -11431.337} C_VEL
LIN {X 0,Y 391.932,Z 258.974,A -85,B 0,C 180,E1 -11431.997,E2 -11431.997} C_VEL
LIN {X 0,Y 392.414,Z 250.928,A -85,B 0,C 180,E1 -11433.851,E2 -11433.851} C_VEL
LIN {X 0,Y 390.369,Z 238.582,A -85,B 0,C 180,E1 -11436.98,E2 -11436.98} C_VEL
LIN {X 0,Y 390.181,Z 238.382,A -85,B 0,C 180,E1 -11440.376,E2 -11440.376} C_VEL
LIN {X 0,Y 390.174,Z 238.381,A -85,B 0,C 180,E1 -11443.542,E2 -11443.542} C_VEL
LIN {X 0,Y 390.136,Z 238.382,A -85,B 0,C 180,E1 -11447.325,E2 -11447.325} C_VEL
LIN {X 0,Y 390.071,Z 238.392,A -85,B 0,C 180,E1 -11451.121,E2 -11451.121} C_VEL
LIN {X 0,Y 390.045,Z 238.394,A -85,B 0,C 180,E1 -11454.483,E2 -11454.483} C_VEL
LIN {X 0,Y 390.073,Z 238.377,A -85,B 0,C 180,E1 -11458.028,E2 -11458.028} C_VEL
LIN {X 0,Y 390.06,Z 238.402,A -85,B 0,C 180,E1 -11461.501,E2 -11461.501} C_VEL
LIN {X 0,Y 390.068,Z 238.388,A -85,B 0,C 180,E1 -11465.208,E2 -11465.208} C_VEL
LIN {X 0,Y 390.076,Z 238.398,A -85,B 0,C 180,E1 -11467.775,E2 -11467.775} C_VEL
LIN {X 0,Y 390.058,Z 238.389,A -85,B 0,C 180,E1 -11470.832,E2 -11470.832} C_VEL
LIN {X 0,Y 390.101,Z 238.384,A -85,B 0,C 180,E1 -11473.903,E2 -11473.903} C_VEL
LIN {X 0,Y 390.087,Z 238.391,A -85,B 0,C 180,E1 -11476.803,E2 -11476.803} C_VEL
LIN {X 0,Y 390.048,Z 238.392,A -85,B 0,C 180,E1 -11479.568,E2 -11479.568} C_VEL
LIN {X 0,Y 390.019,Z 238.388,A -85,B 0,C 180,E1 -11482.453,E2 -11482.453} C_VEL
LIN {X 0,Y 390.042,Z 238.399,A -85,B 0,C 180,E1 -11486.05,E2 -11486.05} C_VEL
LIN {X 0,Y 390.024,Z 238.398,A -85,B 0,C 180,E1 -11488.503,E2 -11488.503} C_VEL
LIN {X 0,Y 390.095,Z 238.369,A -85,B 0,C 180,E1 -11492.075,E2 -11492.075} C_VEL
LIN {X 0,Y 390.061,Z 238.388,A -85,B 0,C 180,E1 -11495.524,E2 -11495.524} C_VEL
LIN {X 0,Y 390.076,Z 238.397,A -85,B 0,C 180,E1 -11498.885,E2 -11498.885} C_VEL
LIN {X 0,Y 390.116,Z 238.377,A -85,B 0,C 180,E1 -11502.172,E2 -11502.172} C_VEL
LIN {X 0,Y 390.135,Z 238.362,A -85,B 0,C 180,E1 -11505.398,E2 -11505.398} C_VEL
LIN {X 0,Y 390.149,Z 238.376,A -85,B 0,C 180,E1 -11508.576,E2 -11508.576} C_VEL
LIN {X 0,Y 390.336,Z 238.359,A -85,B 0,C 180,E1 -11511.998,E2 -11511.998} C_VEL
LIN {X 0,Y 390.222,Z 238.367,A -85,B 0,C 180,E1 -11514.838,E2 -11514.838} C_VEL
LIN {X 0,Y 390.413,Z 238.325,A -85,B 0,C 180,E1 -11517.941,E2 -11517.941} C_VEL
LIN {X 0,Y 390.545,Z 238.324,A -85,B 0,C 180,E1 -11520.005,E2 -11520.005} C_VEL
LIN {X 0,Y 390.308,Z 238.362,A -85,B 0,C 180,E1 -11523.101,E2 -11523.101} C_VEL
LIN {X 0,Y 390.299,Z 238.362,A -85,B 0,C 180,E1 -11526.207,E2 -11526.207} C_VEL
LIN {X 0,Y 390.199,Z 238.359,A -85,B 0,C 180,E1 -11529.333,E2 -11529.333} C_VEL
LIN {X 0,Y 390.173,Z 238.374,A -85,B 0,C 180,E1 -11532.487,E2 -11532.487} C_VEL
LIN {X 0,Y 390.143,Z 238.384,A -85,B 0,C 180,E1 -11535.681,E2 -11535.681} C_VEL
LIN {X 0,Y 390.109,Z 238.379,A -85,B 0,C 180,E1 -11538.926,E2 -11538.926} C_VEL
LIN {X 0,Y 390.043,Z 238.384,A -85,B 0,C 180,E1 -11542.238,E2 -11542.238} C_VEL
LIN {X 0,Y 390.124,Z 238.387,A -85,B 0,C 180,E1 -11545.746,E2 -11545.746} C_VEL
LIN {X 0,Y 390.061,Z 238.384,A -85,B 0,C 180,E1 -11549.113,E2 -11549.113} C_VEL
LIN {X 0,Y 390.049,Z 238.398,A -85,B 0,C 180,E1 -11552.725,E2 -11552.725} C_VEL
LIN {X 0,Y 390.051,Z 238.392,A -85,B 0,C 180,E1 -11555.825,E2 -11555.825} C_VEL
LIN {X 0,Y 390.051,Z 238.398,A -85,B 0,C 180,E1 -11559.216,E2 -11559.216} C_VEL
LIN {X 0,Y 390.047,Z 238.39,A -85,B 0,C 180,E1 -11562.376,E2 -11562.376} C_VEL
LIN {X 0,Y 390.053,Z 238.37,A -85,B 0,C 180,E1 -11565.356,E2 -11565.356} C_VEL
LIN {X 0,Y 390.033,Z 238.398,A -85,B 0,C 180,E1 -11568.188,E2 -11568.188} C_VEL
LIN {X 0,Y 390.069,Z 238.391,A -85,B 0,C 180,E1 -11570.906,E2 -11570.906} C_VEL
LIN {X 0,Y 390.095,Z 238.39,A -85,B 0,C 180,E1 -11574.795,E2 -11574.795} C_VEL
LIN {X 0,Y 390.034,Z 238.398,A -85,B 0,C 180,E1 -11578.497,E2 -11578.497} C_VEL
LIN {X 0,Y 390.13,Z 238.389,A -85,B 0,C 180,E1 -11582.072,E2 -11582.072} C_VEL
LIN {X 0,Y 390.16,Z 238.449,A -85,B 0,C 180,E1 -11582.946,E2 -11582.946} C_VEL
LIN {X 0,Y 390.771,Z 241.496,A -85,B 0,C 180,E1 -11583.76,E2 -11583.76} C_VEL
LIN {X 0,Y 392.757,Z 252.538,A -85,B 0,C 180,E1 -11586.405,E2 -11586.405} C_VEL
LIN {X 0,Y 392.345,Z 260.465,A -85,B 0,C 180,E1 -11588.178,E2 -11588.178} C_VEL
LIN {X 0,Y 391.808,Z 269.049,A -85,B 0,C 180,E1 -11590.023,E2 -11590.023} C_VEL
LIN {X 0,Y 392.473,Z 273.965,A -85,B 0,C 180,E1 -11590.195,E2 -11590.195} C_VEL
LIN {X 0,Y 396.024,Z 297.002,A -85,B 0,C 180,E1 -11590.782,E2 -11590.782} C_VEL
LIN {X 0,Y 394.939,Z 377.06,A -85,B 0,C 180,E1 -11592.258,E2 -11592.258} C_VEL
LIN {X 0,Y 394.366,Z 390.997,A -85,B 0,C 180,E1 -11592.733,E2 -11592.733} C_VEL
LIN {X 0,Y 393.762,Z 402.945,A -85,B 0,C 180,E1 -11593.341,E2 -11593.341} C_VEL
LIN {X 0,Y 392.961,Z 415.028,A -85,B 0,C 180,E1 -11594.173,E2 -11594.173} C_VEL
LIN {X 0,Y 392.18,Z 426.57,A -85,B 0,C 180,E1 -11595.205,E2 -11595.205} C_VEL
LIN {X 0,Y 391.476,Z 436.295,A -85,B 0,C 180,E1 -11596.289,E2 -11596.289} C_VEL
LIN {X 0,Y 390.737,Z 445.445,A -85,B 0,C 180,E1 -11597.536,E2 -11597.536} C_VEL
LIN {X 0,Y 389.944,Z 454.621,A -85,B 0,C 180,E1 -11599.092,E2 -11599.092} C_VEL
LIN {X 0,Y 389.42,Z 462.006,A -85,B 0,C 180,E1 -11600.653,E2 -11600.653} C_VEL
LIN {X 0,Y 389.046,Z 467.918,A -85,B 0,C 180,E1 -11602.214,E2 -11602.214} C_VEL
LIN {X 0,Y 388.787,Z 472.782,A -85,B 0,C 180,E1 -11603.855,E2 -11603.855} C_VEL
LIN {X 0,Y 388.72,Z 476.098,A -85,B 0,C 180,E1 -11605.334,E2 -11605.334} C_VEL
LIN {X 0,Y 388.606,Z 478.61,A -85,B 0,C 180,E1 -11606.89,E2 -11606.89} C_VEL
LIN {X 0,Y 388.622,Z 479.775,A -85,B 0,C 180,E1 -11607.928,E2 -11607.928} C_VEL
LIN {X 0,Y 388.661,Z 480.5,A -85,B 0,C 180,E1 -11608.964,E2 -11608.964} C_VEL
LIN {X 0,Y 388.678,Z 480.837,A -85,B 0,C 180,E1 -11610,E2 -11610} C_VEL
LIN {X 0,Y 388.661,Z 480.789,A -85,B 0,C 180,E1 -11611.036,E2 -11611.036} C_VEL
LIN {X 0,Y 388.621,Z 480.348,A -85,B 0,C 180,E1 -11612.073,E2 -11612.073} C_VEL
LIN {X 0,Y 388.705,Z 478.206,A -85,B 0,C 180,E1 -11614.148,E2 -11614.148} C_VEL
LIN {X 0,Y 388.803,Z 475.242,A -85,B 0,C 180,E1 -11615.843,E2 -11615.843} C_VEL
LIN {X 0,Y 389.117,Z 470.389,A -85,B 0,C 180,E1 -11617.786,E2 -11617.786} C_VEL
LIN {X 0,Y 389.676,Z 464.189,A -85,B 0,C 180,E1 -11619.604,E2 -11619.604} C_VEL
LIN {X 0,Y 390.323,Z 457.455,A -85,B 0,C 180,E1 -11621.161,E2 -11621.161} C_VEL
LIN {X 0,Y 391.227,Z 449.118,A -85,B 0,C 180,E1 -11622.713,E2 -11622.713} C_VEL
LIN {X 0,Y 392.107,Z 440.547,A -85,B 0,C 180,E1 -11624.003,E2 -11624.003} C_VEL
LIN {X 0,Y 393.062,Z 429.832,A -85,B 0,C 180,E1 -11625.313,E2 -11625.313} C_VEL
LIN {X 0,Y 394.1,Z 419.581,A -85,B 0,C 180,E1 -11626.312,E2 -11626.312} C_VEL
LIN {X 0,Y 395.085,Z 408.08,A -85,B 0,C 180,E1 -11627.202,E2 -11627.202} C_VEL
LIN {X 0,Y 395.933,Z 396.175,A -85,B 0,C 180,E1 -11627.897,E2 -11627.897} C_VEL
LIN {X 0,Y 396.658,Z 383.334,A -85,B 0,C 180,E1 -11628.431,E2 -11628.431} C_VEL
LIN {X 0,Y 397.041,Z 370.709,A -85,B 0,C 180,E1 -11628.763,E2 -11628.763} C_VEL
LIN {X 0,Y 398.119,Z 296.336,A -85,B 0,C 180,E1 -11630.147,E2 -11630.147} C_VEL
LIN {X 0,Y 394.222,Z 275.52,A -85,B 0,C 180,E1 -11630.805,E2 -11630.805} C_VEL
LIN {X 0,Y 392.809,Z 268.848,A -85,B 0,C 180,E1 -11631.065,E2 -11631.065} C_VEL
LIN {X 0,Y 393.28,Z 262.968,A -85,B 0,C 180,E1 -11632.318,E2 -11632.318} C_VEL
LIN {X 0,Y 393.701,Z 255.796,A -85,B 0,C 180,E1 -11633.961,E2 -11633.961} C_VEL
LIN {X 0,Y 391.63,Z 245.144,A -85,B 0,C 180,E1 -11636.657,E2 -11636.657} C_VEL
LIN {X 0,Y 390.115,Z 238.472,A -85,B 0,C 180,E1 -11638.487,E2 -11638.487} C_VEL
LIN {X 0,Y 390.045,Z 238.399,A -85,B 0,C 180,E1 -11642.123,E2 -11642.123} C_VEL
LIN {X 0,Y 390.098,Z 238.388,A -85,B 0,C 180,E1 -11645.206,E2 -11645.206} C_VEL
LIN {X 0,Y 390.071,Z 238.388,A -85,B 0,C 180,E1 -11649.095,E2 -11649.095} C_VEL
LIN {X 0,Y 390.049,Z 238.389,A -85,B 0,C 180,E1 -11652.371,E2 -11652.371} C_VEL
LIN {X 0,Y 390.056,Z 238.396,A -85,B 0,C 180,E1 -11655.352,E2 -11655.352} C_VEL
LIN {X 0,Y 390.039,Z 238.386,A -85,B 0,C 180,E1 -11658.184,E2 -11658.184} C_VEL
LIN {X 0,Y 390.075,Z 238.393,A -85,B 0,C 180,E1 -11660.902,E2 -11660.902} C_VEL
LIN {X 0,Y 390.081,Z 238.393,A -85,B 0,C 180,E1 -11664.789,E2 -11664.789} C_VEL
LIN {X 0,Y 390.033,Z 238.395,A -85,B 0,C 180,E1 -11668.493,E2 -11668.493} C_VEL
LIN {X 0,Y 390.026,Z 238.394,A -85,B 0,C 180,E1 -11672,E2 -11672} C_VEL
LIN {X 0,Y 390.052,Z 238.392,A -85,B 0,C 180,E1 -11675.514,E2 -11675.514} C_VEL
LIN {X 0,Y 390.064,Z 238.397,A -85,B 0,C 180,E1 -11678.874,E2 -11678.874} C_VEL
LIN {X 0,Y 390.12,Z 238.388,A -85,B 0,C 180,E1 -11682.162,E2 -11682.162} C_VEL
LIN {X 0,Y 390.151,Z 238.38,A -85,B 0,C 180,E1 -11685.389,E2 -11685.389} C_VEL
LIN {X 0,Y 390.152,Z 238.378,A -85,B 0,C 180,E1 -11688.567,E2 -11688.567} C_VEL
LIN {X 0,Y 390.275,Z 238.369,A -85,B 0,C 180,E1 -11692.068,E2 -11692.068} C_VEL
LIN {X 0,Y 390.216,Z 238.372,A -85,B 0,C 180,E1 -11694.829,E2 -11694.829} C_VEL
LIN {X 0,Y 390.414,Z 238.348,A -85,B 0,C 180,E1 -11697.932,E2 -11697.932} C_VEL
LIN {X 0,Y 390.545,Z 238.336,A -85,B 0,C 180,E1 -11699.995,E2 -11699.995} C_VEL
LIN {X 0,Y 390.277,Z 238.36,A -85,B 0,C 180,E1 -11703.092,E2 -11703.092} C_VEL
LIN {X 0,Y 390.281,Z 238.365,A -85,B 0,C 180,E1 -11706.486,E2 -11706.486} C_VEL
LIN {X 0,Y 390.188,Z 238.379,A -85,B 0,C 180,E1 -11709.324,E2 -11709.324} C_VEL
LIN {X 0,Y 390.164,Z 238.382,A -85,B 0,C 180,E1 -11712.478,E2 -11712.478} C_VEL
LIN {X 0,Y 390.13,Z 238.382,A -85,B 0,C 180,E1 -11715.672,E2 -11715.672} C_VEL
LIN {X 0,Y 390.091,Z 238.391,A -85,B 0,C 180,E1 -11718.917,E2 -11718.917} C_VEL
LIN {X 0,Y 390.026,Z 238.396,A -85,B 0,C 180,E1 -11722.229,E2 -11722.229} C_VEL
LIN {X 0,Y 390.103,Z 238.376,A -85,B 0,C 180,E1 -11725.738,E2 -11725.738} C_VEL
LIN {X 0,Y 390.04,Z 238.401,A -85,B 0,C 180,E1 -11729.104,E2 -11729.104} C_VEL
LIN {X 0,Y 390.021,Z 238.4,A -85,B 0,C 180,E1 -11732.716,E2 -11732.716} C_VEL
LIN {X 0,Y 390.033,Z 238.398,A -85,B 0,C 180,E1 -11735.82,E2 -11735.82} C_VEL
LIN {X 0,Y 390.049,Z 238.397,A -85,B 0,C 180,E1 -11739.214,E2 -11739.214} C_VEL
LIN {X 0,Y 390.093,Z 238.394,A -85,B 0,C 180,E1 -11742.382,E2 -11742.382} C_VEL
LIN {X 0,Y 390.11,Z 238.432,A -85,B 0,C 180,E1 -11745.754,E2 -11745.754} C_VEL
LIN {X 0,Y 390.999,Z 242.495,A -85,B 0,C 180,E1 -11746.919,E2 -11746.919} C_VEL
LIN {X 0,Y 393.044,Z 252.481,A -85,B 0,C 180,E1 -11749.507,E2 -11749.507} C_VEL
LIN {X 0,Y 393.125,Z 257.062,A -85,B 0,C 180,E1 -11750.606,E2 -11750.606} C_VEL
LIN {X 0,Y 393.081,Z 259.223,A -85,B 0,C 180,E1 -11751.008,E2 -11751.008} C_VEL
LIN {X 0,Y 396.956,Z 276.482,A -85,B 0,C 180,E1 -11751.63,E2 -11751.63} C_VEL
LIN {X 0,Y 398.372,Z 285.126,A -85,B 0,C 180,E1 -11751.887,E2 -11751.887} C_VEL
LIN {X 0,Y 396.941,Z 366.838,A -85,B 0,C 180,E1 -11753.423,E2 -11753.423} C_VEL
LIN {X 0,Y 396.392,Z 380.043,A -85,B 0,C 180,E1 -11753.877,E2 -11753.877} C_VEL
LIN {X 0,Y 395.74,Z 391.829,A -85,B 0,C 180,E1 -11754.474,E2 -11754.474} C_VEL
LIN {X 0,Y 394.805,Z 403.677,A -85,B 0,C 180,E1 -11755.275,E2 -11755.275} C_VEL
LIN {X 0,Y 393.89,Z 414.855,A -85,B 0,C 180,E1 -11756.265,E2 -11756.265} C_VEL
LIN {X 0,Y 392.74,Z 426.229,A -85,B 0,C 180,E1 -11757.531,E2 -11757.531} C_VEL
LIN {X 0,Y 391.76,Z 435.992,A -85,B 0,C 180,E1 -11758.908,E2 -11758.908} C_VEL
LIN {X 0,Y 390.856,Z 444.348,A -85,B 0,C 180,E1 -11760.364,E2 -11760.364} C_VEL
LIN {X 0,Y 390.033,Z 452.168,A -85,B 0,C 180,E1 -11762.063,E2 -11762.063} C_VEL
LIN {X 0,Y 389.447,Z 458.244,A -85,B 0,C 180,E1 -11763.76,E2 -11763.76} C_VEL
LIN {X 0,Y 389.055,Z 462.913,A -85,B 0,C 180,E1 -11765.45,E2 -11765.45} C_VEL
LIN {X 0,Y 388.761,Z 466.451,A -85,B 0,C 180,E1 -11767.198,E2 -11767.198} C_VEL
LIN {X 0,Y 388.568,Z 468.614,A -85,B 0,C 180,E1 -11768.793,E2 -11768.793} C_VEL
LIN {X 0,Y 388.53,Z 469.703,A -85,B 0,C 180,E1 -11770.133,E2 -11770.133} C_VEL
LIN {X 0,Y 388.45,Z 470.073,A -85,B 0,C 180,E1 -11772.087,E2 -11772.087} C_VEL
LIN {X 0,Y 388.511,Z 469.515,A -85,B 0,C 180,E1 -11773.46,E2 -11773.46} C_VEL
LIN {X 0,Y 388.544,Z 467.587,A -85,B 0,C 180,E1 -11775.331,E2 -11775.331} C_VEL
LIN {X 0,Y 388.663,Z 465.886,A -85,B 0,C 180,E1 -11776.404,E2 -11776.404} C_VEL
LIN {X 0,Y 388.913,Z 462.456,A -85,B 0,C 180,E1 -11778.005,E2 -11778.005} C_VEL
LIN {X 0,Y 389.116,Z 457.931,A -85,B 0,C 180,E1 -11779.594,E2 -11779.594} C_VEL
LIN {X 0,Y 389.543,Z 452.16,A -85,B 0,C 180,E1 -11781.178,E2 -11781.178} C_VEL
LIN {X 0,Y 390.102,Z 444.911,A -85,B 0,C 180,E1 -11782.755,E2 -11782.755} C_VEL
LIN {X 0,Y 390.793,Z 435.902,A -85,B 0,C 180,E1 -11784.323,E2 -11784.323} C_VEL
LIN {X 0,Y 391.522,Z 426.649,A -85,B 0,C 180,E1 -11785.624,E2 -11785.624} C_VEL
LIN {X 0,Y 392.327,Z 416.33,A -85,B 0,C 180,E1 -11786.791,E2 -11786.791} C_VEL
LIN {X 0,Y 393.165,Z 404.867,A -85,B 0,C 180,E1 -11787.823,E2 -11787.823} C_VEL
LIN {X 0,Y 393.906,Z 392.492,A -85,B 0,C 180,E1 -11788.686,E2 -11788.686} C_VEL
LIN {X 0,Y 394.492,Z 379.771,A -85,B 0,C 180,E1 -11789.33,E2 -11789.33} C_VEL
LIN {X 0,Y 394.966,Z 366.625,A -85,B 0,C 180,E1 -11789.777,E2 -11789.777} C_VEL
LIN {X 0,Y 395.151,Z 353.597,A -85,B 0,C 180,E1 -11790.042,E2 -11790.042} C_VEL
LIN {X 0,Y 394.561,Z 347.789,A -85,B 0,C 180,E1 -11790.174,E2 -11790.174} C_VEL
LIN {X 0,Y 389.332,Z 329.057,A -85,B 0,C 180,E1 -11790.739,E2 -11790.739} C_VEL
LIN {X 0,Y 388.724,Z 323.25,A -85,B 0,C 180,E1 -11790.875,E2 -11790.875} C_VEL
LIN {X 0,Y 389.182,Z 283.126,A -85,B 0,C 180,E1 -11791.623,E2 -11791.623} C_VEL
LIN {X 0,Y 384.999,Z 259.35,A -85,B 0,C 180,E1 -11792.288,E2 -11792.288} C_VEL
LIN {X 0,Y 385.21,Z 255.422,A -85,B 0,C 180,E1 -11793.137,E2 -11793.137} C_VEL
LIN {X 0,Y 385.449,Z 252.154,A -85,B 0,C 180,E1 -11793.92,E2 -11793.92} C_VEL
LIN {X 0,Y 383.339,Z 239.715,A -85,B 0,C 180,E1 -11797.108,E2 -11797.108} C_VEL
LIN {X 0,Y 383.232,Z 239.256,A -85,B 0,C 180,E1 -11797.375,E2 -11797.375} C_VEL
LIN {X 0,Y 383.137,Z 239.261,A -85,B 0,C 180,E1 -11800.569,E2 -11800.569} C_VEL
LIN {X 0,Y 383.105,Z 239.262,A -85,B 0,C 180,E1 -11803.797,E2 -11803.797} C_VEL
LIN {X 0,Y 383.077,Z 239.261,A -85,B 0,C 180,E1 -11807.47,E2 -11807.47} C_VEL
LIN {X 0,Y 383.023,Z 239.263,A -85,B 0,C 180,E1 -11810.665,E2 -11810.665} C_VEL
LIN {X 0,Y 383.007,Z 239.27,A -85,B 0,C 180,E1 -11813.809,E2 -11813.809} C_VEL
LIN {X 0,Y 383.014,Z 239.248,A -85,B 0,C 180,E1 -11817.305,E2 -11817.305} C_VEL
LIN {X 0,Y 382.998,Z 239.275,A -85,B 0,C 180,E1 -11820.917,E2 -11820.917} C_VEL
LIN {X 0,Y 383.015,Z 239.266,A -85,B 0,C 180,E1 -11824.352,E2 -11824.352} C_VEL
LIN {X 0,Y 383.022,Z 239.275,A -85,B 0,C 180,E1 -11827.919,E2 -11827.919} C_VEL
LIN {X 0,Y 383.014,Z 239.268,A -85,B 0,C 180,E1 -11831.343,E2 -11831.343} C_VEL
LIN {X 0,Y 383.051,Z 239.267,A -85,B 0,C 180,E1 -11834.321,E2 -11834.321} C_VEL
LIN {X 0,Y 383.043,Z 239.268,A -85,B 0,C 180,E1 -11837.254,E2 -11837.254} C_VEL
LIN {X 0,Y 382.993,Z 239.258,A -85,B 0,C 180,E1 -11840.417,E2 -11840.417} C_VEL
LIN {X 0,Y 382.999,Z 239.269,A -85,B 0,C 180,E1 -11844.049,E2 -11844.049} C_VEL
LIN {X 0,Y 383.012,Z 239.273,A -85,B 0,C 180,E1 -11847.858,E2 -11847.858} C_VEL
LIN {X 0,Y 383.042,Z 239.247,A -85,B 0,C 180,E1 -11851.725,E2 -11851.725} C_VEL
LIN {X 0,Y 383.033,Z 239.266,A -85,B 0,C 180,E1 -11855.045,E2 -11855.045} C_VEL
LIN {X 0,Y 383.005,Z 239.275,A -85,B 0,C 180,E1 -11858.476,E2 -11858.476} C_VEL
LIN {X 0,Y 383.08,Z 239.253,A -85,B 0,C 180,E1 -11861.833,E2 -11861.833} C_VEL
LIN {X 0,Y 383.099,Z 239.236,A -85,B 0,C 180,E1 -11865.123,E2 -11865.123} C_VEL
LIN {X 0,Y 383.098,Z 239.253,A -85,B 0,C 180,E1 -11868.363,E2 -11868.363} C_VEL
LIN {X 0,Y 383.296,Z 239.236,A -85,B 0,C 180,E1 -11871.938,E2 -11871.938} C_VEL
LIN {X 0,Y 383.194,Z 239.242,A -85,B 0,C 180,E1 -11874.743,E2 -11874.743} C_VEL
LIN {X 0,Y 383.381,Z 239.2,A -85,B 0,C 180,E1 -11877.904,E2 -11877.904} C_VEL
LIN {X 0,Y 383.514,Z 239.198,A -85,B 0,C 180,E1 -11880.005,E2 -11880.005} C_VEL
LIN {X 0,Y 383.244,Z 239.242,A -85,B 0,C 180,E1 -11883.158,E2 -11883.158} C_VEL
LIN {X 0,Y 383.255,Z 239.238,A -85,B 0,C 180,E1 -11886.321,E2 -11886.321} C_VEL
LIN {X 0,Y 383.147,Z 239.237,A -85,B 0,C 180,E1 -11889.507,E2 -11889.507} C_VEL
LIN {X 0,Y 383.128,Z 239.252,A -85,B 0,C 180,E1 -11893.54,E2 -11893.54} C_VEL
LIN {X 0,Y 383.099,Z 239.259,A -85,B 0,C 180,E1 -11897.458,E2 -11897.458} C_VEL
LIN {X 0,Y 383.034,Z 239.254,A -85,B 0,C 180,E1 -11900.65,E2 -11900.65} C_VEL
LIN {X 0,Y 383.028,Z 239.267,A -85,B 0,C 180,E1 -11903.812,E2 -11903.812} C_VEL
LIN {X 0,Y 383.086,Z 239.265,A -85,B 0,C 180,E1 -11906.127,E2 -11906.127} C_VEL
LIN {X 0,Y 382.996,Z 239.259,A -85,B 0,C 180,E1 -11909.703,E2 -11909.703} C_VEL
LIN {X 0,Y 383.007,Z 239.277,A -85,B 0,C 180,E1 -11913.404,E2 -11913.404} C_VEL
LIN {X 0,Y 383.031,Z 239.266,A -85,B 0,C 180,E1 -11916.165,E2 -11916.165} C_VEL
LIN {X 0,Y 382.997,Z 239.275,A -85,B 0,C 180,E1 -11919.964,E2 -11919.964} C_VEL
LIN {X 0,Y 383.016,Z 239.267,A -85,B 0,C 180,E1 -11922.781,E2 -11922.781} C_VEL
LIN {X 0,Y 383.006,Z 239.25,A -85,B 0,C 180,E1 -11925.791,E2 -11925.791} C_VEL
LIN {X 0,Y 382.976,Z 239.276,A -85,B 0,C 180,E1 -11928.802,E2 -11928.802} C_VEL
LIN {X 0,Y 383.004,Z 239.269,A -85,B 0,C 180,E1 -11932.1,E2 -11932.1} C_VEL
LIN {X 0,Y 383.029,Z 239.272,A -85,B 0,C 180,E1 -11935.334,E2 -11935.334} C_VEL
LIN {X 0,Y 382.993,Z 239.277,A -85,B 0,C 180,E1 -11939.083,E2 -11939.083} C_VEL
LIN {X 0,Y 383.124,Z 239.297,A -85,B 0,C 180,E1 -11942.704,E2 -11942.704} C_VEL
LIN {X 0,Y 383.554,Z 241.455,A -85,B 0,C 180,E1 -11943.321,E2 -11943.321} C_VEL
LIN {X 0,Y 385.802,Z 253.989,A -85,B 0,C 180,E1 -11946.374,E2 -11946.374} C_VEL
LIN {X 0,Y 385.031,Z 266.23,A -85,B 0,C 180,E1 -11949.15,E2 -11949.15} C_VEL
LIN {X 0,Y 384.894,Z 269.103,A -85,B 0,C 180,E1 -11949.728,E2 -11949.728} C_VEL
LIN {X 0,Y 389.217,Z 297.854,A -85,B 0,C 180,E1 -11950.505,E2 -11950.505} C_VEL
LIN {X 0,Y 388.074,Z 377.275,A -85,B 0,C 180,E1 -11952.001,E2 -11952.001} C_VEL
LIN {X 0,Y 387.494,Z 391.116,A -85,B 0,C 180,E1 -11952.485,E2 -11952.485} C_VEL
LIN {X 0,Y 386.821,Z 404.061,A -85,B 0,C 180,E1 -11953.169,E2 -11953.169} C_VEL
LIN {X 0,Y 385.973,Z 415.852,A -85,B 0,C 180,E1 -11954.014,E2 -11954.014} C_VEL
LIN {X 0,Y 385.175,Z 427.234,A -85,B 0,C 180,E1 -11955.065,E2 -11955.065} C_VEL
LIN {X 0,Y 384.388,Z 437.472,A -85,B 0,C 180,E1 -11956.25,E2 -11956.25} C_VEL
LIN {X 0,Y 383.604,Z 446.67,A -85,B 0,C 180,E1 -11957.569,E2 -11957.569} C_VEL
LIN {X 0,Y 382.848,Z 455.623,A -85,B 0,C 180,E1 -11959.155,E2 -11959.155} C_VEL
LIN {X 0,Y 382.303,Z 462.802,A -85,B 0,C 180,E1 -11960.744,E2 -11960.744} C_VEL
LIN {X 0,Y 381.879,Z 469.324,A -85,B 0,C 180,E1 -11962.599,E2 -11962.599} C_VEL
LIN {X 0,Y 381.701,Z 472.897,A -85,B 0,C 180,E1 -11963.88,E2 -11963.88} C_VEL
LIN {X 0,Y 381.626,Z 476.844,A -85,B 0,C 180,E1 -11965.776,E2 -11965.776} C_VEL
LIN {X 0,Y 381.521,Z 478.442,A -85,B 0,C 180,E1 -11966.832,E2 -11966.832} C_VEL
LIN {X 0,Y 381.52,Z 479.633,A -85,B 0,C 180,E1 -11967.889,E2 -11967.889} C_VEL
LIN {X 0,Y 381.56,Z 480.379,A -85,B 0,C 180,E1 -11968.945,E2 -11968.945} C_VEL
LIN {X 0,Y 381.579,Z 480.731,A -85,B 0,C 180,E1 -11970,E2 -11970} C_VEL
LIN {X 0,Y 381.559,Z 480.698,A -85,B 0,C 180,E1 -11971.056,E2 -11971.056} C_VEL
LIN {X 0,Y 381.519,Z 480.279,A -85,B 0,C 180,E1 -11972.112,E2 -11972.112} C_VEL
LIN {X 0,Y 381.635,Z 478.175,A -85,B 0,C 180,E1 -11974.225,E2 -11974.225} C_VEL
LIN {X 0,Y 381.752,Z 474.763,A -85,B 0,C 180,E1 -11976.191,E2 -11976.191} C_VEL
LIN {X 0,Y 382.077,Z 470.446,A -85,B 0,C 180,E1 -11977.93,E2 -11977.93} C_VEL
LIN {X 0,Y 382.646,Z 464.301,A -85,B 0,C 180,E1 -11979.782,E2 -11979.782} C_VEL
LIN {X 0,Y 383.331,Z 457.621,A -85,B 0,C 180,E1 -11981.367,E2 -11981.367} C_VEL
LIN {X 0,Y 384.317,Z 449.348,A -85,B 0,C 180,E1 -11982.945,E2 -11982.945} C_VEL
LIN {X 0,Y 385.231,Z 440.864,A -85,B 0,C 180,E1 -11984.258,E2 -11984.258} C_VEL
LIN {X 0,Y 386.235,Z 430.373,A -85,B 0,C 180,E1 -11985.574,E2 -11985.574} C_VEL
LIN {X 0,Y 387.45,Z 418.669,A -85,B 0,C 180,E1 -11986.736,E2 -11986.736} C_VEL
LIN {X 0,Y 388.513,Z 406.853,A -85,B 0,C 180,E1 -11987.638,E2 -11987.638} C_VEL
LIN {X 0,Y 389.39,Z 394.604,A -85,B 0,C 180,E1 -11988.344,E2 -11988.344} C_VEL
LIN {X 0,Y 390.126,Z 382.071,A -85,B 0,C 180,E1 -11988.853,E2 -11988.853} C_VEL
LIN {X 0,Y 390.522,Z 368.412,A -85,B 0,C 180,E1 -11989.19,E2 -11989.19} C_VEL
LIN {X 0,Y 391.616,Z 297.413,A -85,B 0,C 180,E1 -11990.534,E2 -11990.534} C_VEL
LIN {X 0,Y 387.849,Z 277.128,A -85,B 0,C 180,E1 -11991.195,E2 -11991.195} C_VEL
LIN {X 0,Y 385.995,Z 268.663,A -85,B 0,C 180,E1 -11991.53,E2 -11991.53} C_VEL
LIN {X 0,Y 386.87,Z 258.491,A -85,B 0,C 180,E1 -11993.817,E2 -11993.817} C_VEL
LIN {X 0,Y 385.711,Z 251.287,A -85,B 0,C 180,E1 -11995.642,E2 -11995.642} C_VEL
LIN {X 0,Y 383.398,Z 240.693,A -85,B 0,C 180,E1 -11998.464,E2 -11998.464} C_VEL
LIN {X 0,Y 383.054,Z 239.3,A -85,B 0,C 180,E1 -11998.941,E2 -11998.941} C_VEL
LIN {X 0,Y 383,Z 239.274,A -85,B 0,C 180,E1 -12002.421,E2 -12002.421} C_VEL
LIN {X 0,Y 383.037,Z 239.267,A -85,B 0,C 180,E1 -12005.954,E2 -12005.954} C_VEL
LIN {X 0,Y 382.999,Z 239.271,A -85,B 0,C 180,E1 -12009.579,E2 -12009.579} C_VEL
LIN {X 0,Y 383.02,Z 239.264,A -85,B 0,C 180,E1 -12012.777,E2 -12012.777} C_VEL
LIN {X 0,Y 383.009,Z 239.274,A -85,B 0,C 180,E1 -12015.787,E2 -12015.787} C_VEL
LIN {X 0,Y 382.997,Z 239.271,A -85,B 0,C 180,E1 -12018.794,E2 -12018.794} C_VEL
LIN {X 0,Y 383.007,Z 239.271,A -85,B 0,C 180,E1 -12022.095,E2 -12022.095} C_VEL
LIN {X 0,Y 383.023,Z 239.273,A -85,B 0,C 180,E1 -12025.329,E2 -12025.329} C_VEL
LIN {X 0,Y 382.993,Z 239.278,A -85,B 0,C 180,E1 -12029.078,E2 -12029.078} C_VEL
LIN {X 0,Y 382.981,Z 239.274,A -85,B 0,C 180,E1 -12032.688,E2 -12032.688} C_VEL
LIN {X 0,Y 383.019,Z 239.266,A -85,B 0,C 180,E1 -12036.188,E2 -12036.188} C_VEL
LIN {X 0,Y 383.065,Z 239.261,A -85,B 0,C 180,E1 -12039.595,E2 -12039.595} C_VEL
LIN {X 0,Y 383.102,Z 239.263,A -85,B 0,C 180,E1 -12042.927,E2 -12042.927} C_VEL
LIN {X 0,Y 383.133,Z 239.257,A -85,B 0,C 180,E1 -12046.46,E2 -12046.46} C_VEL
LIN {X 0,Y 383.148,Z 239.255,A -85,B 0,C 180,E1 -12050.493,E2 -12050.493} C_VEL
LIN {X 0,Y 383.264,Z 239.238,A -85,B 0,C 180,E1 -12053.679,E2 -12053.679} C_VEL
LIN {X 0,Y 383.38,Z 239.224,A -85,B 0,C 180,E1 -12057.894,E2 -12057.894} C_VEL
LIN {X 0,Y 383.514,Z 239.211,A -85,B 0,C 180,E1 -12059.995,E2 -12059.995} C_VEL
LIN {X 0,Y 383.215,Z 239.239,A -85,B 0,C 180,E1 -12063.149,E2 -12063.149} C_VEL
LIN {X 0,Y 383.244,Z 239.241,A -85,B 0,C 180,E1 -12066.473,E2 -12066.473} C_VEL
LIN {X 0,Y 383.138,Z 239.257,A -85,B 0,C 180,E1 -12069.497,E2 -12069.497} C_VEL
LIN {X 0,Y 383.118,Z 239.26,A -85,B 0,C 180,E1 -12073.531,E2 -12073.531} C_VEL
LIN {X 0,Y 383.084,Z 239.266,A -85,B 0,C 180,E1 -12077.064,E2 -12077.064} C_VEL
LIN {X 0,Y 383.017,Z 239.277,A -85,B 0,C 180,E1 -12080.642,E2 -12080.642} C_VEL
LIN {X 0,Y 383.019,Z 239.272,A -85,B 0,C 180,E1 -12083.802,E2 -12083.802} C_VEL
LIN {X 0,Y 383.063,Z 239.251,A -85,B 0,C 180,E1 -12086.118,E2 -12086.118} C_VEL
LIN {X 0,Y 382.973,Z 239.275,A -85,B 0,C 180,E1 -12089.695,E2 -12089.695} C_VEL
LIN {X 0,Y 382.981,Z 239.28,A -85,B 0,C 180,E1 -12093.395,E2 -12093.395} C_VEL
LIN {X 0,Y 383.01,Z 239.275,A -85,B 0,C 180,E1 -12096.16,E2 -12096.16} C_VEL
LIN {X 0,Y 382.994,Z 239.277,A -85,B 0,C 180,E1 -12099.952,E2 -12099.952} C_VEL
LIN {X 0,Y 383.037,Z 239.271,A -85,B 0,C 180,E1 -12102.783,E2 -12102.783} C_VEL
LIN {X 0,Y 383.057,Z 239.402,A -85,B 0,C 180,E1 -12105.402,E2 -12105.402} C_VEL
LIN {X 0,Y 385.411,Z 250.247,A -85,B 0,C 180,E1 -12108.376,E2 -12108.376} C_VEL
LIN {X 0,Y 386.37,Z 255.78,A -85,B 0,C 180,E1 -12109.805,E2 -12109.805} C_VEL
LIN {X 0,Y 386.283,Z 259.027,A -85,B 0,C 180,E1 -12110.524,E2 -12110.524} C_VEL
LIN {X 0,Y 388.727,Z 269.274,A -85,B 0,C 180,E1 -12110.943,E2 -12110.943} C_VEL
LIN {X 0,Y 391.825,Z 284.893,A -85,B 0,C 180,E1 -12111.466,E2 -12111.466} C_VEL
LIN {X 0,Y 390.367,Z 367.194,A -85,B 0,C 180,E1 -12113.047,E2 -12113.047} C_VEL
LIN {X 0,Y 389.764,Z 380.678,A -85,B 0,C 180,E1 -12113.523,E2 -12113.523} C_VEL
LIN {X 0,Y 389.025,Z 393.058,A -85,B 0,C 180,E1 -12114.172,E2 -12114.172} C_VEL
LIN {X 0,Y 387.99,Z 405.36,A -85,B 0,C 180,E1 -12115.051,E2 -12115.051} C_VEL
LIN {X 0,Y 387.022,Z 416.201,A -85,B 0,C 180,E1 -12116.051,E2 -12116.051} C_VEL
LIN {X 0,Y 385.986,Z 426.235,A -85,B 0,C 180,E1 -12117.201,E2 -12117.201} C_VEL
LIN {X 0,Y 384.891,Z 436.274,A -85,B 0,C 180,E1 -12118.641,E2 -12118.641} C_VEL
LIN {X 0,Y 383.95,Z 444.379,A -85,B 0,C 180,E1 -12120.079,E2 -12120.079} C_VEL
LIN {X 0,Y 383.131,Z 451.71,A -85,B 0,C 180,E1 -12121.687,E2 -12121.687} C_VEL
LIN {X 0,Y 382.525,Z 457.401,A -85,B 0,C 180,E1 -12123.248,E2 -12123.248} C_VEL
LIN {X 0,Y 382.081,Z 462.31,A -85,B 0,C 180,E1 -12124.972,E2 -12124.972} C_VEL
LIN {X 0,Y 381.718,Z 466.444,A -85,B 0,C 180,E1 -12126.992,E2 -12126.992} C_VEL
LIN {X 0,Y 381.502,Z 468.398,A -85,B 0,C 180,E1 -12128.38,E2 -12128.38} C_VEL
LIN {X 0,Y 381.446,Z 469.769,A -85,B 0,C 180,E1 -12129.972,E2 -12129.972} C_VEL
LIN {X 0,Y 381.351,Z 470.218,A -85,B 0,C 180,E1 -12131.742,E2 -12131.742} C_VEL
LIN {X 0,Y 381.408,Z 469.682,A -85,B 0,C 180,E1 -12133.345,E2 -12133.345} C_VEL
LIN {X 0,Y 381.419,Z 468.087,A -85,B 0,C 180,E1 -12135.05,E2 -12135.05} C_VEL
LIN {X 0,Y 381.613,Z 465.534,A -85,B 0,C 180,E1 -12136.69,E2 -12136.69} C_VEL
LIN {X 0,Y 381.848,Z 461.939,A -85,B 0,C 180,E1 -12138.319,E2 -12138.319} C_VEL
LIN {X 0,Y 382.094,Z 457.213,A -85,B 0,C 180,E1 -12139.936,E2 -12139.936} C_VEL
LIN {X 0,Y 382.709,Z 450.105,A -85,B 0,C 180,E1 -12141.805,E2 -12141.805} C_VEL
LIN {X 0,Y 383.279,Z 442.325,A -85,B 0,C 180,E1 -12143.419,E2 -12143.419} C_VEL
LIN {X 0,Y 383.903,Z 434.396,A -85,B 0,C 180,E1 -12144.748,E2 -12144.748} C_VEL
LIN {X 0,Y 384.695,Z 424.706,A -85,B 0,C 180,E1 -12146.071,E2 -12146.071} C_VEL
LIN {X 0,Y 385.595,Z 413.923,A -85,B 0,C 180,E1 -12147.257,E2 -12147.257} C_VEL
LIN {X 0,Y 386.337,Z 403.824,A -85,B 0,C 180,E1 -12148.148,E2 -12148.148} C_VEL
LIN {X 0,Y 387.039,Z 392.114,A -85,B 0,C 180,E1 -12148.959,E2 -12148.959} C_VEL
LIN {X 0,Y 387.66,Z 379.298,A -85,B 0,C 180,E1 -12149.61,E2 -12149.61} C_VEL
LIN {X 0,Y 388.118,Z 366.11,A -85,B 0,C 180,E1 -12150.058,E2 -12150.058} C_VEL
LIN {X 0,Y 388.724,Z 323.25,A -85,B 0,C 180,E1 -12150.875,E2 -12150.875} C_VEL
LIN {X 0,Y 388.105,Z 317.437,A -85,B 0,C 180,E1 -12151.012,E2 -12151.012} C_VEL
LIN {X 0,Y 382.871,Z 298.702,A -85,B 0,C 180,E1 -12151.598,E2 -12151.598} C_VEL
LIN {X 0,Y 382.361,Z 292.887,A -85,B 0,C 180,E1 -12151.733,E2 -12151.733} C_VEL
LIN {X 0,Y 382.33,Z 283.772,A -85,B 0,C 180,E1 -12151.912,E2 -12151.912} C_VEL
LIN {X 0,Y 378.118,Z 259.698,A -85,B 0,C 180,E1 -12152.597,E2 -12152.597} C_VEL
LIN {X 0,Y 378.062,Z 258.724,A -85,B 0,C 180,E1 -12152.717,E2 -12152.717} C_VEL
LIN {X 0,Y 378.466,Z 253.381,A -85,B 0,C 180,E1 -12153.993,E2 -12153.993} C_VEL
LIN {X 0,Y 376.574,Z 241.937,A -85,B 0,C 180,E1 -12156.967,E2 -12156.967} C_VEL
LIN {X 0,Y 376.204,Z 240.168,A -85,B 0,C 180,E1 -12157.514,E2 -12157.514} C_VEL
LIN {X 0,Y 376.084,Z 240.141,A -85,B 0,C 180,E1 -12160.77,E2 -12160.77} C_VEL
LIN {X 0,Y 376.043,Z 240.143,A -85,B 0,C 180,E1 -12164.061,E2 -12164.061} C_VEL
LIN {X 0,Y 376.045,Z 240.136,A -85,B 0,C 180,E1 -12167.632,E2 -12167.632} C_VEL
LIN {X 0,Y 375.996,Z 240.14,A -85,B 0,C 180,E1 -12170.86,E2 -12170.86} C_VEL
LIN {X 0,Y 375.96,Z 240.148,A -85,B 0,C 180,E1 -12174.283,E2 -12174.283} C_VEL
LIN {X 0,Y 375.977,Z 240.123,A -85,B 0,C 180,E1 -12176.655,E2 -12176.655} C_VEL
LIN {X 0,Y 375.966,Z 240.148,A -85,B 0,C 180,E1 -12180.312,E2 -12180.312} C_VEL
LIN {X 0,Y 375.967,Z 240.153,A -85,B 0,C 180,E1 -12182.826,E2 -12182.826} C_VEL
LIN {X 0,Y 375.988,Z 240.143,A -85,B 0,C 180,E1 -12186.521,E2 -12186.521} C_VEL
LIN {X 0,Y 375.979,Z 240.147,A -85,B 0,C 180,E1 -12189.98,E2 -12189.98} C_VEL
LIN {X 0,Y 375.975,Z 240.141,A -85,B 0,C 180,E1 -12193.759,E2 -12193.759} C_VEL
LIN {X 0,Y 375.971,Z 240.149,A -85,B 0,C 180,E1 -12196.804,E2 -12196.804} C_VEL
LIN {X 0,Y 375.97,Z 240.138,A -85,B 0,C 180,E1 -12200.032,E2 -12200.032} C_VEL
LIN {X 0,Y 375.938,Z 240.144,A -85,B 0,C 180,E1 -12203.5,E2 -12203.5} C_VEL
LIN {X 0,Y 375.935,Z 240.154,A -85,B 0,C 180,E1 -12205.894,E2 -12205.894} C_VEL
LIN {X 0,Y 375.946,Z 240.145,A -85,B 0,C 180,E1 -12209.693,E2 -12209.693} C_VEL
LIN {X 0,Y 375.981,Z 240.125,A -85,B 0,C 180,E1 -12212.147,E2 -12212.147} C_VEL
LIN {X 0,Y 375.986,Z 240.135,A -85,B 0,C 180,E1 -12214.544,E2 -12214.544} C_VEL
LIN {X 0,Y 375.967,Z 240.149,A -85,B 0,C 180,E1 -12218.052,E2 -12218.052} C_VEL
LIN {X 0,Y 376.017,Z 240.134,A -85,B 0,C 180,E1 -12221.48,E2 -12221.48} C_VEL
LIN {X 0,Y 376.047,Z 240.112,A -85,B 0,C 180,E1 -12224.838,E2 -12224.838} C_VEL
LIN {X 0,Y 376.049,Z 240.131,A -85,B 0,C 180,E1 -12228.142,E2 -12228.142} C_VEL
LIN {X 0,Y 376.25,Z 240.114,A -85,B 0,C 180,E1 -12231.882,E2 -12231.882} C_VEL
LIN {X 0,Y 376.166,Z 240.116,A -85,B 0,C 180,E1 -12234.645,E2 -12234.645} C_VEL
LIN {X 0,Y 376.347,Z 240.075,A -85,B 0,C 180,E1 -12237.865,E2 -12237.865} C_VEL
LIN {X 0,Y 376.484,Z 240.073,A -85,B 0,C 180,E1 -12240.005,E2 -12240.005} C_VEL
LIN {X 0,Y 376.183,Z 240.122,A -85,B 0,C 180,E1 -12243.218,E2 -12243.218} C_VEL
LIN {X 0,Y 376.213,Z 240.114,A -85,B 0,C 180,E1 -12246.44,E2 -12246.44} C_VEL
LIN {X 0,Y 376.117,Z 240.11,A -85,B 0,C 180,E1 -12249.686,E2 -12249.686} C_VEL
LIN {X 0,Y 376.092,Z 240.129,A -85,B 0,C 180,E1 -12253.662,E2 -12253.662} C_VEL
LIN {X 0,Y 376.048,Z 240.138,A -85,B 0,C 180,E1 -12257.611,E2 -12257.611} C_VEL
LIN {X 0,Y 375.984,Z 240.131,A -85,B 0,C 180,E1 -12260.836,E2 -12260.836} C_VEL
LIN {X 0,Y 375.993,Z 240.146,A -85,B 0,C 180,E1 -12264.286,E2 -12264.286} C_VEL
LIN {X 0,Y 376.026,Z 240.148,A -85,B 0,C 180,E1 -12266.656,E2 -12266.656} C_VEL
LIN {X 0,Y 375.971,Z 240.136,A -85,B 0,C 180,E1 -12270.316,E2 -12270.316} C_VEL
LIN {X 0,Y 375.966,Z 240.152,A -85,B 0,C 180,E1 -12274.115,E2 -12274.115} C_VEL
LIN {X 0,Y 375.958,Z 240.147,A -85,B 0,C 180,E1 -12276.745,E2 -12276.745} C_VEL
LIN {X 0,Y 375.979,Z 240.149,A -85,B 0,C 180,E1 -12279.97,E2 -12279.97} C_VEL
LIN {X 0,Y 375.938,Z 240.133,A -85,B 0,C 180,E1 -12283.769,E2 -12283.769} C_VEL
LIN {X 0,Y 375.945,Z 240.139,A -85,B 0,C 180,E1 -12286.813,E2 -12286.813} C_VEL
LIN {X 0,Y 375.946,Z 240.15,A -85,B 0,C 180,E1 -12290.536,E2 -12290.536} C_VEL
LIN {X 0,Y 375.974,Z 240.15,A -85,B 0,C 180,E1 -12293.498,E2 -12293.498} C_VEL
LIN {X 0,Y 375.971,Z 240.148,A -85,B 0,C 180,E1 -12295.89,E2 -12295.89} C_VEL
LIN {X 0,Y 375.975,Z 240.154,A -85,B 0,C 180,E1 -12299.689,E2 -12299.689} C_VEL
LIN {X 0,Y 376.108,Z 240.274,A -85,B 0,C 180,E1 -12302.529,E2 -12302.529} C_VEL
LIN {X 0,Y 378.58,Z 253.565,A -85,B 0,C 180,E1 -12305.896,E2 -12305.896} C_VEL
LIN {X 0,Y 378.791,Z 257.28,A -85,B 0,C 180,E1 -12306.78,E2 -12306.78} C_VEL
LIN {X 0,Y 377.895,Z 268.753,A -85,B 0,C 180,E1 -12309.379,E2 -12309.379} C_VEL
LIN {X 0,Y 378.809,Z 274.768,A -85,B 0,C 180,E1 -12309.584,E2 -12309.584} C_VEL
LIN {X 0,Y 382.4,Z 298.795,A -85,B 0,C 180,E1 -12310.22,E2 -12310.22} C_VEL
LIN {X 0,Y 381.246,Z 376.269,A -85,B 0,C 180,E1 -12311.702,E2 -12311.702} C_VEL
LIN {X 0,Y 380.683,Z 389.651,A -85,B 0,C 180,E1 -12312.161,E2 -12312.161} C_VEL
LIN {X 0,Y 379.996,Z 401.897,A -85,B 0,C 180,E1 -12312.788,E2 -12312.788} C_VEL
LIN {X 0,Y 379.253,Z 413.431,A -85,B 0,C 180,E1 -12313.585,E2 -12313.585} C_VEL
LIN {X 0,Y 378.459,Z 423.947,A -85,B 0,C 180,E1 -12314.518,E2 -12314.518} C_VEL
LIN {X 0,Y 377.704,Z 434.378,A -85,B 0,C 180,E1 -12315.677,E2 -12315.677} C_VEL
LIN {X 0,Y 376.782,Z 444.496,A -85,B 0,C 180,E1 -12317.066,E2 -12317.066} C_VEL
LIN {X 0,Y 376.032,Z 452.454,A -85,B 0,C 180,E1 -12318.41,E2 -12318.41} C_VEL
LIN {X 0,Y 375.444,Z 460.218,A -85,B 0,C 180,E1 -12320.029,E2 -12320.029} C_VEL
LIN {X 0,Y 374.913,Z 467.348,A -85,B 0,C 180,E1 -12321.918,E2 -12321.918} C_VEL
LIN {X 0,Y 374.643,Z 472.08,A -85,B 0,C 180,E1 -12323.538,E2 -12323.538} C_VEL
LIN {X 0,Y 374.559,Z 475.686,A -85,B 0,C 180,E1 -12325.157,E2 -12325.157} C_VEL
LIN {X 0,Y 374.439,Z 478.267,A -85,B 0,C 180,E1 -12326.772,E2 -12326.772} C_VEL
LIN {X 0,Y 374.42,Z 479.48,A -85,B 0,C 180,E1 -12327.849,E2 -12327.849} C_VEL
LIN {X 0,Y 374.459,Z 480.255,A -85,B 0,C 180,E1 -12328.925,E2 -12328.925} C_VEL
LIN {X 0,Y 374.48,Z 480.624,A -85,B 0,C 180,E1 -12330,E2 -12330} C_VEL
LIN {X 0,Y 374.458,Z 480.607,A -85,B 0,C 180,E1 -12331.076,E2 -12331.076} C_VEL
LIN {X 0,Y 374.419,Z 480.208,A -85,B 0,C 180,E1 -12332.152,E2 -12332.152} C_VEL
LIN {X 0,Y 374.44,Z 479.389,A -85,B 0,C 180,E1 -12333.228,E2 -12333.228} C_VEL
LIN {X 0,Y 374.565,Z 478.155,A -85,B 0,C 180,E1 -12334.305,E2 -12334.305} C_VEL
LIN {X 0,Y 374.654,Z 475.095,A -85,B 0,C 180,E1 -12336.149,E2 -12336.149} C_VEL
LIN {X 0,Y 375.035,Z 470.506,A -85,B 0,C 180,E1 -12338.08,E2 -12338.08} C_VEL
LIN {X 0,Y 375.634,Z 464.419,A -85,B 0,C 180,E1 -12339.966,E2 -12339.966} C_VEL
LIN {X 0,Y 376.355,Z 457.786,A -85,B 0,C 180,E1 -12341.581,E2 -12341.581} C_VEL
LIN {X 0,Y 377.415,Z 449.568,A -85,B 0,C 180,E1 -12343.186,E2 -12343.186} C_VEL
LIN {X 0,Y 378.367,Z 441.169,A -85,B 0,C 180,E1 -12344.523,E2 -12344.523} C_VEL
LIN {X 0,Y 379.383,Z 431.061,A -85,B 0,C 180,E1 -12345.83,E2 -12345.83} C_VEL
LIN {X 0,Y 380.575,Z 420.617,A -85,B 0,C 180,E1 -12346.909,E2 -12346.909} C_VEL
LIN {X 0,Y 381.647,Z 409.473,A -85,B 0,C 180,E1 -12347.828,E2 -12347.828} C_VEL
LIN {X 0,Y 382.543,Z 398.206,A -85,B 0,C 180,E1 -12348.546,E2 -12348.546} C_VEL
LIN {X 0,Y 383.364,Z 385.47,A -85,B 0,C 180,E1 -12349.129,E2 -12349.129} C_VEL
LIN {X 0,Y 383.878,Z 372.416,A -85,B 0,C 180,E1 -12349.512,E2 -12349.512} C_VEL
LIN {X 0,Y 385.15,Z 298.267,A -85,B 0,C 180,E1 -12350.944,E2 -12350.944} C_VEL
LIN {X 0,Y 381.003,Z 276.42,A -85,B 0,C 180,E1 -12351.681,E2 -12351.681} C_VEL
LIN {X 0,Y 379.217,Z 268.484,A -85,B 0,C 180,E1 -12352.016,E2 -12352.016} C_VEL
LIN {X 0,Y 380.018,Z 259.81,A -85,B 0,C 180,E1 -12354.008,E2 -12354.008} C_VEL
LIN {X 0,Y 378.324,Z 250.361,A -85,B 0,C 180,E1 -12356.477,E2 -12356.477} C_VEL
LIN {X 0,Y 376.037,Z 240.455,A -85,B 0,C 180,E1 -12359.227,E2 -12359.227} C_VEL
LIN {X 0,Y 375.972,Z 240.154,A -85,B 0,C 180,E1 -12359.694,E2 -12359.694} C_VEL
LIN {X 0,Y 375.964,Z 240.148,A -85,B 0,C 180,E1 -12362.827,E2 -12362.827} C_VEL
LIN {X 0,Y 375.97,Z 240.147,A -85,B 0,C 180,E1 -12365.414,E2 -12365.414} C_VEL
LIN {X 0,Y 375.948,Z 240.148,A -85,B 0,C 180,E1 -12368.261,E2 -12368.261} C_VEL
LIN {X 0,Y 375.932,Z 240.154,A -85,B 0,C 180,E1 -12371.596,E2 -12371.596} C_VEL
LIN {X 0,Y 375.939,Z 240.158,A -85,B 0,C 180,E1 -12374.729,E2 -12374.729} C_VEL
LIN {X 0,Y 375.945,Z 240.143,A -85,B 0,C 180,E1 -12378.398,E2 -12378.398} C_VEL
LIN {X 0,Y 375.958,Z 240.155,A -85,B 0,C 180,E1 -12380.533,E2 -12380.533} C_VEL
LIN {X 0,Y 375.971,Z 240.15,A -85,B 0,C 180,E1 -12383.494,E2 -12383.494} C_VEL
LIN {X 0,Y 375.969,Z 240.15,A -85,B 0,C 180,E1 -12385.886,E2 -12385.886} C_VEL
LIN {X 0,Y 375.973,Z 240.151,A -85,B 0,C 180,E1 -12389.684,E2 -12389.684} C_VEL
LIN {X 0,Y 375.928,Z 240.15,A -85,B 0,C 180,E1 -12392.132,E2 -12392.132} C_VEL
LIN {X 0,Y 375.946,Z 240.154,A -85,B 0,C 180,E1 -12394.531,E2 -12394.531} C_VEL
LIN {X 0,Y 375.984,Z 240.146,A -85,B 0,C 180,E1 -12396.883,E2 -12396.883} C_VEL
LIN {X 0,Y 376.006,Z 240.139,A -85,B 0,C 180,E1 -12400.336,E2 -12400.336} C_VEL
LIN {X 0,Y 376.033,Z 240.137,A -85,B 0,C 180,E1 -12403.715,E2 -12403.715} C_VEL
LIN {X 0,Y 376.11,Z 240.134,A -85,B 0,C 180,E1 -12407.038,E2 -12407.038} C_VEL
LIN {X 0,Y 376.118,Z 240.132,A -85,B 0,C 180,E1 -12410.314,E2 -12410.314} C_VEL
LIN {X 0,Y 376.223,Z 240.115,A -85,B 0,C 180,E1 -12413.56,E2 -12413.56} C_VEL
LIN {X 0,Y 376.345,Z 240.101,A -85,B 0,C 180,E1 -12417.855,E2 -12417.855} C_VEL
LIN {X 0,Y 376.484,Z 240.087,A -85,B 0,C 180,E1 -12419.995,E2 -12419.995} C_VEL
LIN {X 0,Y 376.345,Z 240.101,A -85,B 0,C 180,E1 -12422.136,E2 -12422.136} C_VEL
LIN {X 0,Y 376.214,Z 240.117,A -85,B 0,C 180,E1 -12426.455,E2 -12426.455} C_VEL
LIN {X 0,Y 376.108,Z 240.134,A -85,B 0,C 180,E1 -12429.676,E2 -12429.676} C_VEL
LIN {X 0,Y 376.082,Z 240.136,A -85,B 0,C 180,E1 -12433.652,E2 -12433.652} C_VEL
LIN {X 0,Y 376.022,Z 240.144,A -85,B 0,C 180,E1 -12437.394,E2 -12437.394} C_VEL
LIN {X 0,Y 375.966,Z 240.154,A -85,B 0,C 180,E1 -12440.827,E2 -12440.827} C_VEL
LIN {X 0,Y 375.979,Z 240.15,A -85,B 0,C 180,E1 -12444.276,E2 -12444.276} C_VEL
LIN {X 0,Y 376.003,Z 240.131,A -85,B 0,C 180,E1 -12446.647,E2 -12446.647} C_VEL
LIN {X 0,Y 375.945,Z 240.148,A -85,B 0,C 180,E1 -12450.307,E2 -12450.307} C_VEL
LIN {X 0,Y 375.937,Z 240.153,A -85,B 0,C 180,E1 -12454.106,E2 -12454.106} C_VEL
LIN {X 0,Y 375.935,Z 240.157,A -85,B 0,C 180,E1 -12456.735,E2 -12456.735} C_VEL
LIN {X 0,Y 375.973,Z 240.152,A -85,B 0,C 180,E1 -12459.968,E2 -12459.968} C_VEL
LIN {X 0,Y 375.97,Z 240.15,A -85,B 0,C 180,E1 -12463.195,E2 -12463.195} C_VEL
LIN {X 0,Y 376.058,Z 240.365,A -85,B 0,C 180,E1 -12465.016,E2 -12465.016} C_VEL
LIN {X 0,Y 378.432,Z 251.201,A -85,B 0,C 180,E1 -12468.043,E2 -12468.043} C_VEL
LIN {X 0,Y 379.502,Z 257.93,A -85,B 0,C 180,E1 -12469.813,E2 -12469.813} C_VEL
LIN {X 0,Y 379.524,Z 259.28,A -85,B 0,C 180,E1 -12470.064,E2 -12470.064} C_VEL
LIN {X 0,Y 383.661,Z 277.037,A -85,B 0,C 180,E1 -12470.756,E2 -12470.756} C_VEL
LIN {X 0,Y 385.39,Z 286.589,A -85,B 0,C 180,E1 -12471.071,E2 -12471.071} C_VEL
LIN {X 0,Y 383.831,Z 366.812,A -85,B 0,C 180,E1 -12472.63,E2 -12472.63} C_VEL
LIN {X 0,Y 383.248,Z 379.88,A -85,B 0,C 180,E1 -12473.089,E2 -12473.089} C_VEL
LIN {X 0,Y 382.46,Z 392.344,A -85,B 0,C 180,E1 -12473.738,E2 -12473.738} C_VEL
LIN {X 0,Y 381.519,Z 403.651,A -85,B 0,C 180,E1 -12474.531,E2 -12474.531} C_VEL
LIN {X 0,Y 380.474,Z 414.843,A -85,B 0,C 180,E1 -12475.549,E2 -12475.549} C_VEL
LIN {X 0,Y 379.224,Z 426.243,A -85,B 0,C 180,E1 -12476.858,E2 -12476.858} C_VEL
LIN {X 0,Y 378.068,Z 436.292,A -85,B 0,C 180,E1 -12478.322,E2 -12478.322} C_VEL
LIN {X 0,Y 377.055,Z 444.41,A -85,B 0,C 180,E1 -12479.784,E2 -12479.784} C_VEL
LIN {X 0,Y 376.19,Z 451.645,A -85,B 0,C 180,E1 -12481.394,E2 -12481.394} C_VEL
LIN {X 0,Y 375.632,Z 456.479,A -85,B 0,C 180,E1 -12482.716,E2 -12482.716} C_VEL
LIN {X 0,Y 375.106,Z 461.633,A -85,B 0,C 180,E1 -12484.473,E2 -12484.473} C_VEL
LIN {X 0,Y 374.747,Z 465.484,A -85,B 0,C 180,E1 -12486.221,E2 -12486.221} C_VEL
LIN {X 0,Y 374.461,Z 468.153,A -85,B 0,C 180,E1 -12487.953,E2 -12487.953} C_VEL
LIN {X 0,Y 374.354,Z 469.836,A -85,B 0,C 180,E1 -12489.81,E2 -12489.81} C_VEL
LIN {X 0,Y 374.254,Z 470.318,A -85,B 0,C 180,E1 -12491.383,E2 -12491.383} C_VEL
LIN {X 0,Y 374.304,Z 469.831,A -85,B 0,C 180,E1 -12493.227,E2 -12493.227} C_VEL
LIN {X 0,Y 374.32,Z 468.508,A -85,B 0,C 180,E1 -12494.76,E2 -12494.76} C_VEL
LIN {X 0,Y 374.404,Z 467.052,A -85,B 0,C 180,E1 -12495.875,E2 -12495.875} C_VEL
LIN {X 0,Y 374.616,Z 464.543,A -85,B 0,C 180,E1 -12497.269,E2 -12497.269} C_VEL
LIN {X 0,Y 374.889,Z 459.849,A -85,B 0,C 180,E1 -12499.195,E2 -12499.195} C_VEL
LIN {X 0,Y 375.337,Z 453.478,A -85,B 0,C 180,E1 -12501.113,E2 -12501.113} C_VEL
LIN {X 0,Y 375.922,Z 446.54,A -85,B 0,C 180,E1 -12502.75,E2 -12502.75} C_VEL
LIN {X 0,Y 376.508,Z 439.464,A -85,B 0,C 180,E1 -12504.107,E2 -12504.107} C_VEL
LIN {X 0,Y 377.176,Z 430.948,A -85,B 0,C 180,E1 -12505.458,E2 -12505.458} C_VEL
LIN {X 0,Y 378.092,Z 420.379,A -85,B 0,C 180,E1 -12506.803,E2 -12506.803} C_VEL
LIN {X 0,Y 378.997,Z 409.88,A -85,B 0,C 180,E1 -12507.874,E2 -12507.874} C_VEL
LIN {X 0,Y 379.828,Z 398.201,A -85,B 0,C 180,E1 -12508.819,E2 -12508.819} C_VEL
LIN {X 0,Y 380.466,Z 385.256,A -85,B 0,C 180,E1 -12509.603,E2 -12509.603} C_VEL
LIN {X 0,Y 381.073,Z 371.883,A -85,B 0,C 180,E1 -12510.165,E2 -12510.165} C_VEL
LIN {X 0,Y 381.391,Z 357.041,A -85,B 0,C 180,E1 -12510.528,E2 -12510.528} C_VEL
LIN {X 0,Y 382.361,Z 292.887,A -85,B 0,C 180,E1 -12511.733,E2 -12511.733} C_VEL
LIN {X 0,Y 381.67,Z 289.09,A -85,B 0,C 180,E1 -12511.838,E2 -12511.838} C_VEL
LIN {X 0,Y 378.493,Z 283.449,A -85,B 0,C 180,E1 -12512.091,E2 -12512.091} C_VEL
LIN {X 0,Y 374.919,Z 277.873,A -85,B 0,C 180,E1 -12512.367,E2 -12512.367} C_VEL
LIN {X 0,Y 373.646,Z 274.125,A -85,B 0,C 180,E1 -12512.502,E2 -12512.502} C_VEL
LIN {X 0,Y 371.156,Z 259.536,A -85,B 0,C 180,E1 -12512.951,E2 -12512.951} C_VEL
LIN {X 0,Y 371.211,Z 257.881,A -85,B 0,C 180,E1 -12513.256,E2 -12513.256} C_VEL
LIN {X 0,Y 371.484,Z 254.609,A -85,B 0,C 180,E1 -12514.068,E2 -12514.068} C_VEL
LIN {X 0,Y 369.573,Z 243.166,A -85,B 0,C 180,E1 -12517.1,E2 -12517.1} C_VEL
LIN {X 0,Y 369.144,Z 241.032,A -85,B 0,C 180,E1 -12517.766,E2 -12517.766} C_VEL
LIN {X 0,Y 369.022,Z 241.02,A -85,B 0,C 180,E1 -12520.979,E2 -12520.979} C_VEL
LIN {X 0,Y 368.986,Z 241.02,A -85,B 0,C 180,E1 -12524.336,E2 -12524.336} C_VEL
LIN {X 0,Y 368.99,Z 241.014,A -85,B 0,C 180,E1 -12527.787,E2 -12527.787} C_VEL
LIN {X 0,Y 368.944,Z 241.024,A -85,B 0,C 180,E1 -12531.218,E2 -12531.218} C_VEL
LIN {X 0,Y 368.92,Z 241.019,A -85,B 0,C 180,E1 -12534.778,E2 -12534.778} C_VEL
LIN {X 0,Y 368.948,Z 241.007,A -85,B 0,C 180,E1 -12538.438,E2 -12538.438} C_VEL
LIN {X 0,Y 368.911,Z 241.031,A -85,B 0,C 180,E1 -12542.236,E2 -12542.236} C_VEL
LIN {X 0,Y 368.927,Z 241.023,A -85,B 0,C 180,E1 -12546.195,E2 -12546.195} C_VEL
LIN {X 0,Y 368.943,Z 241.026,A -85,B 0,C 180,E1 -12548.947,E2 -12548.947} C_VEL
LIN {X 0,Y 368.908,Z 241.016,A -85,B 0,C 180,E1 -12552.024,E2 -12552.024} C_VEL
LIN {X 0,Y 368.969,Z 241.019,A -85,B 0,C 180,E1 -12555.199,E2 -12555.199} C_VEL
LIN {X 0,Y 368.915,Z 241.027,A -85,B 0,C 180,E1 -12558.191,E2 -12558.191} C_VEL
LIN {X 0,Y 368.884,Z 241.011,A -85,B 0,C 180,E1 -12561.364,E2 -12561.364} C_VEL
LIN {X 0,Y 368.91,Z 241.027,A -85,B 0,C 180,E1 -12565.151,E2 -12565.151} C_VEL
LIN {X 0,Y 368.905,Z 241.023,A -85,B 0,C 180,E1 -12569.052,E2 -12569.052} C_VEL
LIN {X 0,Y 368.965,Z 240.999,A -85,B 0,C 180,E1 -12571.57,E2 -12571.57} C_VEL
LIN {X 0,Y 368.94,Z 241.02,A -85,B 0,C 180,E1 -12575.23,E2 -12575.23} C_VEL
LIN {X 0,Y 368.954,Z 241.027,A -85,B 0,C 180,E1 -12578.965,E2 -12578.965} C_VEL
LIN {X 0,Y 368.978,Z 241.01,A -85,B 0,C 180,E1 -12582.263,E2 -12582.263} C_VEL
LIN {X 0,Y 369.026,Z 240.992,A -85,B 0,C 180,E1 -12586.233,E2 -12586.233} C_VEL
LIN {X 0,Y 369.064,Z 241.008,A -85,B 0,C 180,E1 -12590.137,E2 -12590.137} C_VEL
LIN {X 0,Y 369.181,Z 240.993,A -85,B 0,C 180,E1 -12592.347,E2 -12592.347} C_VEL
LIN {X 0,Y 369.139,Z 240.991,A -85,B 0,C 180,E1 -12594.543,E2 -12594.543} C_VEL
LIN {X 0,Y 369.312,Z 240.951,A -85,B 0,C 180,E1 -12597.824,E2 -12597.824} C_VEL
LIN {X 0,Y 369.453,Z 240.948,A -85,B 0,C 180,E1 -12600.005,E2 -12600.005} C_VEL
LIN {X 0,Y 369.314,Z 240.979,A -85,B 0,C 180,E1 -12602.186,E2 -12602.186} C_VEL
LIN {X 0,Y 369.173,Z 240.99,A -85,B 0,C 180,E1 -12606.563,E2 -12606.563} C_VEL
LIN {X 0,Y 369.066,Z 240.987,A -85,B 0,C 180,E1 -12609.873,E2 -12609.873} C_VEL
LIN {X 0,Y 369.04,Z 241.008,A -85,B 0,C 180,E1 -12613.776,E2 -12613.776} C_VEL
LIN {X 0,Y 369.006,Z 241.016,A -85,B 0,C 180,E1 -12617.772,E2 -12617.772} C_VEL
LIN {X 0,Y 368.915,Z 241.011,A -85,B 0,C 180,E1 -12621.225,E2 -12621.225} C_VEL
LIN {X 0,Y 368.96,Z 241.028,A -85,B 0,C 180,E1 -12624.779,E2 -12624.779} C_VEL
LIN {X 0,Y 368.97,Z 241.021,A -85,B 0,C 180,E1 -12627.207,E2 -12627.207} C_VEL
LIN {X 0,Y 368.919,Z 241.021,A -85,B 0,C 180,E1 -12630.991,E2 -12630.991} C_VEL
LIN {X 0,Y 368.939,Z 241.032,A -85,B 0,C 180,E1 -12634.857,E2 -12634.857} C_VEL
LIN {X 0,Y 368.889,Z 241.028,A -85,B 0,C 180,E1 -12638.637,E2 -12638.637} C_VEL
LIN {X 0,Y 368.888,Z 241.026,A -85,B 0,C 180,E1 -12642.011,E2 -12642.011} C_VEL
LIN {X 0,Y 368.888,Z 241.003,A -85,B 0,C 180,E1 -12645.178,E2 -12645.178} C_VEL
LIN {X 0,Y 368.882,Z 241.033,A -85,B 0,C 180,E1 -12648.178,E2 -12648.178} C_VEL
LIN {X 0,Y 368.888,Z 241.028,A -85,B 0,C 180,E1 -12651.368,E2 -12651.368} C_VEL
LIN {X 0,Y 368.948,Z 241.025,A -85,B 0,C 180,E1 -12655.148,E2 -12655.148} C_VEL
LIN {X 0,Y 368.925,Z 241.029,A -85,B 0,C 180,E1 -12659.047,E2 -12659.047} C_VEL
LIN {X 0,Y 369.027,Z 241.126,A -85,B 0,C 180,E1 -12662.264,E2 -12662.264} C_VEL
LIN {X 0,Y 370.063,Z 246.498,A -85,B 0,C 180,E1 -12663.706,E2 -12663.706} C_VEL
LIN {X 0,Y 371.718,Z 255.623,A -85,B 0,C 180,E1 -12666.016,E2 -12666.016} C_VEL
LIN {X 0,Y 371.622,Z 260.545,A -85,B 0,C 180,E1 -12667.19,E2 -12667.19} C_VEL
LIN {X 0,Y 370.995,Z 268.85,A -85,B 0,C 180,E1 -12669.068,E2 -12669.068} C_VEL
LIN {X 0,Y 373.591,Z 286.197,A -85,B 0,C 180,E1 -12669.572,E2 -12669.572} C_VEL
LIN {X 0,Y 375.581,Z 299.375,A -85,B 0,C 180,E1 -12669.925,E2 -12669.925} C_VEL
LIN {X 0,Y 374.408,Z 376.433,A -85,B 0,C 180,E1 -12671.427,E2 -12671.427} C_VEL
LIN {X 0,Y 373.834,Z 389.72,A -85,B 0,C 180,E1 -12671.894,E2 -12671.894} C_VEL
LIN {X 0,Y 373.113,Z 401.92,A -85,B 0,C 180,E1 -12672.531,E2 -12672.531} C_VEL
LIN {X 0,Y 372.277,Z 414.234,A -85,B 0,C 180,E1 -12673.41,E2 -12673.41} C_VEL
LIN {X 0,Y 371.469,Z 424.57,A -85,B 0,C 180,E1 -12674.36,E2 -12674.36} C_VEL
LIN {X 0,Y 370.687,Z 434.786,A -85,B 0,C 180,E1 -12675.528,E2 -12675.528} C_VEL
LIN {X 0,Y 369.805,Z 443.996,A -85,B 0,C 180,E1 -12676.818,E2 -12676.818} C_VEL
LIN {X 0,Y 369.057,Z 452.024,A -85,B 0,C 180,E1 -12678.188,E2 -12678.188} C_VEL
LIN {X 0,Y 368.403,Z 459.869,A -85,B 0,C 180,E1 -12679.837,E2 -12679.837} C_VEL
LIN {X 0,Y 367.871,Z 467.048,A -85,B 0,C 180,E1 -12681.763,E2 -12681.763} C_VEL
LIN {X 0,Y 367.577,Z 471.824,A -85,B 0,C 180,E1 -12683.413,E2 -12683.413} C_VEL
LIN {X 0,Y 367.459,Z 475.47,A -85,B 0,C 180,E1 -12685.063,E2 -12685.063} C_VEL
LIN {X 0,Y 367.359,Z 478.089,A -85,B 0,C 180,E1 -12686.71,E2 -12686.71} C_VEL
LIN {X 0,Y 367.324,Z 479.32,A -85,B 0,C 180,E1 -12687.807,E2 -12687.807} C_VEL
LIN {X 0,Y 367.357,Z 480.129,A -85,B 0,C 180,E1 -12688.904,E2 -12688.904} C_VEL
LIN {X 0,Y 367.381,Z 480.516,A -85,B 0,C 180,E1 -12690,E2 -12690} C_VEL
LIN {X 0,Y 367.356,Z 480.517,A -85,B 0,C 180,E1 -12691.097,E2 -12691.097} C_VEL
LIN {X 0,Y 367.323,Z 480.135,A -85,B 0,C 180,E1 -12692.193,E2 -12692.193} C_VEL
LIN {X 0,Y 367.361,Z 479.351,A -85,B 0,C 180,E1 -12693.291,E2 -12693.291} C_VEL
LIN {X 0,Y 367.474,Z 478.135,A -85,B 0,C 180,E1 -12694.388,E2 -12694.388} C_VEL
LIN {X 0,Y 367.553,Z 475.434,A -85,B 0,C 180,E1 -12696.102,E2 -12696.102} C_VEL
LIN {X 0,Y 367.981,Z 470.561,A -85,B 0,C 180,E1 -12698.236,E2 -12698.236} C_VEL
LIN {X 0,Y 368.533,Z 465.514,A -85,B 0,C 180,E1 -12699.883,E2 -12699.883} C_VEL
LIN {X 0,Y 369.27,Z 459.19,A -85,B 0,C 180,E1 -12701.528,E2 -12701.528} C_VEL
LIN {X 0,Y 370.295,Z 451.293,A -85,B 0,C 180,E1 -12703.165,E2 -12703.165} C_VEL
LIN {X 0,Y 371.496,Z 441.623,A -85,B 0,C 180,E1 -12704.778,E2 -12704.778} C_VEL
LIN {X 0,Y 372.568,Z 431.53,A -85,B 0,C 180,E1 -12706.127,E2 -12706.127} C_VEL
LIN {X 0,Y 373.833,Z 421.206,A -85,B 0,C 180,E1 -12707.224,E2 -12707.224} C_VEL
LIN {X 0,Y 374.949,Z 410.224,A -85,B 0,C 180,E1 -12708.157,E2 -12708.157} C_VEL
LIN {X 0,Y 375.975,Z 398.073,A -85,B 0,C 180,E1 -12708.953,E2 -12708.953} C_VEL
LIN {X 0,Y 376.828,Z 385.318,A -85,B 0,C 180,E1 -12709.545,E2 -12709.545} C_VEL
LIN {X 0,Y 377.375,Z 371.939,A -85,B 0,C 180,E1 -12709.941,E2 -12709.941} C_VEL
LIN {X 0,Y 378.712,Z 299.426,A -85,B 0,C 180,E1 -12711.361,E2 -12711.361} C_VEL
LIN {X 0,Y 374.608,Z 277.699,A -85,B 0,C 180,E1 -12712.112,E2 -12712.112} C_VEL
LIN {X 0,Y 372.498,Z 268.488,A -85,B 0,C 180,E1 -12712.508,E2 -12712.508} C_VEL
LIN {X 0,Y 373.082,Z 262.423,A -85,B 0,C 180,E1 -12713.892,E2 -12713.892} C_VEL
LIN {X 0,Y 372.711,Z 258.489,A -85,B 0,C 180,E1 -12714.902,E2 -12714.902} C_VEL
LIN {X 0,Y 370.409,Z 247.113,A -85,B 0,C 180,E1 -12718.008,E2 -12718.008} C_VEL
LIN {X 0,Y 368.949,Z 241.072,A -85,B 0,C 180,E1 -12719.825,E2 -12719.825} C_VEL
LIN {X 0,Y 368.911,Z 241.028,A -85,B 0,C 180,E1 -12723.537,E2 -12723.537} C_VEL
LIN {X 0,Y 368.913,Z 241.033,A -85,B 0,C 180,E1 -12726.853,E2 -12726.853} C_VEL
LIN {X 0,Y 368.897,Z 241.035,A -85,B 0,C 180,E1 -12730.372,E2 -12730.372} C_VEL
LIN {X 0,Y 368.895,Z 241.027,A -85,B 0,C 180,E1 -12733.614,E2 -12733.614} C_VEL
LIN {X 0,Y 368.898,Z 241.018,A -85,B 0,C 180,E1 -12736.693,E2 -12736.693} C_VEL
LIN {X 0,Y 368.922,Z 241.029,A -85,B 0,C 180,E1 -12739.641,E2 -12739.641} C_VEL
LIN {X 0,Y 368.909,Z 241.032,A -85,B 0,C 180,E1 -12743.143,E2 -12743.143} C_VEL
LIN {X 0,Y 368.907,Z 241.033,A -85,B 0,C 180,E1 -12746.459,E2 -12746.459} C_VEL
LIN {X 0,Y 368.908,Z 241.031,A -85,B 0,C 180,E1 -12749.04,E2 -12749.04} C_VEL
LIN {X 0,Y 368.918,Z 241.023,A -85,B 0,C 180,E1 -12751.555,E2 -12751.555} C_VEL
LIN {X 0,Y 368.897,Z 241.028,A -85,B 0,C 180,E1 -12755.216,E2 -12755.216} C_VEL
LIN {X 0,Y 368.93,Z 241.03,A -85,B 0,C 180,E1 -12757.601,E2 -12757.601} C_VEL
LIN {X 0,Y 368.963,Z 241.02,A -85,B 0,C 180,E1 -12761.102,E2 -12761.102} C_VEL
LIN {X 0,Y 369.005,Z 241.008,A -85,B 0,C 180,E1 -12764.531,E2 -12764.531} C_VEL
LIN {X 0,Y 369.01,Z 241.015,A -85,B 0,C 180,E1 -12767.902,E2 -12767.902} C_VEL
LIN {X 0,Y 369.151,Z 241.002,A -85,B 0,C 180,E1 -12771.887,E2 -12771.887} C_VEL
LIN {X 0,Y 369.133,Z 240.999,A -85,B 0,C 180,E1 -12774.533,E2 -12774.533} C_VEL
LIN {X 0,Y 369.309,Z 240.977,A -85,B 0,C 180,E1 -12777.814,E2 -12777.814} C_VEL
LIN {X 0,Y 369.453,Z 240.962,A -85,B 0,C 180,E1 -12779.995,E2 -12779.995} C_VEL
LIN {X 0,Y 369.309,Z 240.977,A -85,B 0,C 180,E1 -12782.176,E2 -12782.176} C_VEL
